C03569=1018.076,43.871,-109.128,166.538,54.047,159.849
C03570=1018.081,44.120,-109.143,166.541,54.040,159.848
C03571=1018.087,44.370,-109.159,166.544,54.032,159.847
C03572=1018.092,44.619,-109.174,166.546,54.025,159.846
C03573=1018.097,44.868,-109.190,166.549,54.018,159.846
C03574=1018.102,45.118,-109.206,166.552,54.011,159.845
C03575=1018.107,45.367,-109.221,166.553,54.004,159.844
C03576=1018.113,45.617,-109.237,166.556,53.997,159.843
C03577=1018.118,45.867,-109.252,166.559,53.989,159.842
C03578=1018.123,46.116,-109.267,166.561,53.982,159.841
C03579=1018.129,46.365,-109.283,166.564,53.975,159.841
C03580=1018.134,46.615,-109.298,166.567,53.968,159.840
C03581=1018.140,46.865,-109.314,166.569,53.961,159.839
C03582=1018.145,47.114,-109.329,166.572,53.954,159.838
C03583=1018.150,47.364,-109.345,166.575,53.946,159.837
C03584=1018.156,47.612,-109.361,166.577,53.939,159.836
C03585=1018.161,47.862,-109.376,166.580,53.932,159.836
C03586=1018.166,48.112,-109.391,166.582,53.925,159.835
C03587=1018.171,48.361,-109.406,166.584,53.918,159.834
C03588=1018.177,48.610,-109.423,166.587,53.911,159.833
C03589=1018.182,48.860,-109.438,166.590,53.903,159.832
C03590=1018.188,49.110,-109.453,166.592,53.896,159.831
C03591=1018.193,49.359,-109.469,166.595,53.889,159.831
C03592=1018.199,49.608,-109.485,166.598,53.882,159.830
C03593=1018.203,49.858,-109.501,166.600,53.875,159.829
C03594=1018.209,50.108,-109.516,166.603,53.868,159.828
C03595=1018.214,50.357,-109.531,166.606,53.860,159.827
C03596=1018.220,50.606,-109.548,166.609,53.853,159.827
C03597=1018.225,50.856,-109.563,166.611,53.846,159.826
C03598=1018.231,51.106,-109.578,166.613,53.839,159.825
C03599=1018.236,51.354,-109.594,166.616,53.832,159.824
C03600=1018.242,51.604,-109.610,166.618,53.825,159.823
C03601=1018.247,51.853,-109.625,166.621,53.817,159.822
C03602=1018.253,52.103,-109.641,166.624,53.810,159.821
C03603=1018.258,52.352,-109.656,166.626,53.803,159.820
C03604=1018.263,52.602,-109.672,166.629,53.795,159.820
C03605=1018.268,52.851,-109.687,166.632,53.788,159.819
C03606=1018.274,53.101,-109.703,166.634,53.781,159.818
C03607=1018.279,53.350,-109.719,166.636,53.774,159.817
C03608=1018.285,53.600,-109.735,166.639,53.767,159.816
C03609=1018.290,53.849,-109.751,166.642,53.759,159.815
C03610=1018.295,54.099,-109.766,166.645,53.752,159.815
C03611=1018.301,54.347,-109.782,166.647,53.745,159.814
C03612=1018.306,54.597,-109.798,166.650,53.737,159.813
C03613=1018.312,54.847,-109.813,166.653,53.730,159.812
C03614=1018.317,55.096,-109.829,166.655,53.723,159.811
C03615=1018.323,55.346,-109.845,166.657,53.715,159.810
C03616=1018.328,55.595,-109.860,166.660,53.708,159.809
C03617=1018.334,55.845,-109.876,166.663,53.701,159.809
C03618=1018.339,56.094,-109.891,166.665,53.694,159.808
C03619=1018.345,56.343,-109.907,166.668,53.687,159.807
C03620=1018.351,56.593,-109.923,166.670,53.679,159.806
C03621=1018.356,56.842,-109.939,166.673,53.671,159.805
C03622=1018.361,57.092,-109.955,166.675,53.665,159.804
C03623=1018.366,57.341,-109.971,166.678,53.657,159.803
C03624=1018.372,57.591,-109.986,166.681,53.650,159.803
C03625=1018.377,57.841,-110.002,166.684,53.642,159.802
C03626=1018.383,58.089,-110.018,166.687,53.635,159.801
C03627=1018.388,58.339,-110.033,166.689,53.628,159.800
C03628=1018.395,58.621,-110.051,166.692,53.620,159.799
C03629=1018.401,58.904,-110.069,166.694,53.611,159.798
C03630=1018.407,59.186,-110.088,166.698,53.603,159.797
C03631=1018.413,59.469,-110.105,166.700,53.595,159.796
C03632=1018.419,59.718,-110.121,166.703,53.587,159.795
C03633=1018.425,59.968,-110.137,166.706,53.580,159.794
C03634=1018.430,60.217,-110.153,166.709,53.572,159.793
C03635=1018.436,60.467,-110.168,166.712,53.565,159.792
C03636=1018.441,60.715,-110.184,166.714,53.558,159.792
C03637=1018.447,60.965,-110.200,166.716,53.550,159.791
C03638=1018.453,61.215,-110.216,166.719,53.543,159.790
C03639=1018.458,61.464,-110.231,166.722,53.536,159.789
C03640=1018.463,61.714,-110.248,166.725,53.528,159.788
C03641=1018.469,61.964,-110.263,166.727,53.521,159.787
C03642=1018.474,62.213,-110.280,166.730,53.514,159.786
C03643=1018.480,62.462,-110.296,166.732,53.506,159.785
C03644=1018.485,62.712,-110.311,166.735,53.499,159.784
C03645=1018.491,62.961,-110.327,166.738,53.491,159.784
C03646=1018.496,63.211,-110.343,166.740,53.485,159.783
C03647=1018.502,63.460,-110.359,166.743,53.477,159.782
C03648=1018.507,63.701,-110.376,166.745,53.470,159.781
C03649=1018.512,63.942,-110.391,166.748,53.463,159.780
C03650=1018.518,64.183,-110.407,166.750,53.456,159.779
C03651=1018.523,64.424,-110.422,166.753,53.449,159.779
C03652=1018.528,64.666,-110.438,166.756,53.442,159.778
C03653=1018.533,64.907,-110.454,166.758,53.435,159.777
C03654=1018.539,65.148,-110.469,166.761,53.428,159.776
C03655=1018.543,65.389,-110.485,166.763,53.421,159.775
C03656=1018.549,65.638,-110.501,166.766,53.414,159.774
C03657=1018.554,65.888,-110.518,166.768,53.407,159.773
C03658=1018.560,66.137,-110.534,166.770,53.399,159.772
C03659=1018.565,66.387,-110.550,166.773,53.392,159.772
C03660=1018.571,66.636,-110.566,166.777,53.385,159.771
C03661=1018.576,66.885,-110.582,166.778,53.378,159.770
C03662=1018.581,67.135,-110.599,166.781,53.371,159.769
C03663=1018.587,67.384,-110.615,166.785,53.363,159.768
C03664=1018.592,67.634,-110.631,166.786,53.356,159.767
C03665=1018.597,67.883,-110.647,166.789,53.349,159.766
C03666=1018.603,68.133,-110.664,166.792,53.342,159.766
C03667=1018.609,68.382,-110.680,166.795,53.334,159.765
C03668=1018.614,68.632,-110.697,166.797,53.327,159.764
C03669=1018.619,68.880,-110.713,166.800,53.320,159.763
C03670=1018.624,69.130,-110.730,166.803,53.312,159.762
C03671=1018.630,69.380,-110.747,166.805,53.306,159.761
C03672=1018.635,69.629,-110.763,166.808,53.298,159.761
C03673=1018.640,69.878,-110.779,166.811,53.291,159.760
C03674=1018.646,70.127,-110.796,166.813,53.284,159.759
C03675=1018.651,70.377,-110.813,166.816,53.277,159.758
C03676=1018.656,70.627,-110.829,166.818,53.269,159.757
C03677=1018.662,70.876,-110.846,166.820,53.262,159.756
C03678=1018.667,71.125,-110.862,166.823,53.255,159.755
C03679=1018.673,71.374,-110.878,166.826,53.248,159.755
C03680=1018.678,71.624,-110.895,166.828,53.241,159.754
C03681=1018.683,71.874,-110.912,166.831,53.234,159.753
C03682=1018.689,72.123,-110.928,166.834,53.226,159.752
C03683=1018.694,72.372,-110.945,166.836,53.219,159.751
C03684=1018.699,72.621,-110.962,166.839,53.212,159.750
C03685=1018.705,72.871,-110.978,166.842,53.205,159.749
C03686=1018.710,73.120,-110.995,166.845,53.198,159.749
C03687=1018.716,73.370,-111.012,166.847,53.190,159.747
C03688=1018.721,73.619,-111.028,166.850,53.183,159.747
C03689=1018.726,73.868,-111.044,166.853,53.176,159.746
C03690=1018.732,74.118,-111.061,166.855,53.169,159.745
C03691=1018.737,74.367,-111.078,166.858,53.162,159.744
C03692=1018.743,74.666,-111.098,166.861,53.153,159.743
C03693=1018.750,74.965,-111.118,166.864,53.144,159.742
C03694=1018.756,75.265,-111.138,166.868,53.136,159.741
C03695=1018.763,75.563,-111.158,166.871,53.127,159.740
C03696=1018.768,75.813,-111.175,166.873,53.120,159.739
C03697=1018.774,76.062,-111.191,166.876,53.112,159.738
C03698=1018.780,76.312,-111.208,166.879,53.105,159.737
C03699=1018.785,76.560,-111.225,166.881,53.098,159.736
C03700=1018.790,76.810,-111.242,166.884,53.091,159.736
C03701=1018.796,77.059,-111.258,166.887,53.084,159.735
C03702=1018.801,77.309,-111.275,166.888,53.076,159.734
C03703=1018.806,77.559,-111.292,166.891,53.069,159.733
C03704=1018.812,77.808,-111.309,166.894,53.062,159.732
C03705=1018.817,78.057,-111.326,166.897,53.055,159.731
C03706=1018.822,78.307,-111.343,166.900,53.048,159.730
C03707=1018.828,78.556,-111.360,166.903,53.041,159.730
C03708=1018.832,78.805,-111.377,166.905,53.034,159.729
C03709=1018.837,79.055,-111.394,166.908,53.027,159.728
C03710=1018.843,79.304,-111.411,166.910,53.019,159.727
C03711=1018.848,79.553,-111.428,166.912,53.012,159.726
C03712=1018.854,79.803,-111.444,166.915,53.005,159.725
C03713=1018.860,80.052,-111.462,166.919,52.998,159.725
C03714=1018.865,80.301,-111.479,166.921,52.991,159.724
C03715=1018.870,80.551,-111.496,166.924,52.984,159.723
C03716=1018.876,80.800,-111.513,166.927,52.977,159.722
C03717=1018.881,81.050,-111.530,166.928,52.969,159.721
C03718=1018.886,81.299,-111.547,166.931,52.962,159.720
C03719=1018.891,81.548,-111.564,166.934,52.955,159.719
C03720=1018.896,81.797,-111.581,166.937,52.948,159.718
C03721=1018.902,82.046,-111.599,166.940,52.941,159.718
C03722=1018.907,82.296,-111.615,166.942,52.933,159.717
C03723=1018.912,82.546,-111.632,166.944,52.927,159.716
C03724=1018.918,82.795,-111.650,166.947,52.919,159.715
C03725=1018.923,83.044,-111.667,166.950,52.912,159.714
C03726=1018.928,83.293,-111.684,166.953,52.905,159.713
C03727=1018.934,83.543,-111.701,166.955,52.898,159.712
C03728=1018.939,83.792,-111.717,166.958,52.890,159.712
C03729=1018.945,84.041,-111.735,166.961,52.883,159.711
C03730=1018.950,84.291,-111.752,166.963,52.877,159.710
C03731=1018.956,84.540,-111.769,166.966,52.869,159.709
C03732=1018.961,84.790,-111.786,166.969,52.862,159.708
C03733=1018.966,85.039,-111.804,166.971,52.855,159.707
C03734=1018.972,85.289,-111.821,166.974,52.848,159.706
C03735=1018.977,85.538,-111.838,166.977,52.840,159.705
C03736=1018.982,85.787,-111.855,166.980,52.833,159.705
C03737=1018.988,86.036,-111.873,166.982,52.826,159.704
C03738=1018.993,86.286,-111.890,166.985,52.819,159.703
C03739=1018.998,86.536,-111.906,166.988,52.811,159.702
C03740=1019.004,86.785,-111.924,166.990,52.804,159.701
C03741=1019.009,87.034,-111.941,166.993,52.797,159.700
C03742=1019.015,87.283,-111.958,166.996,52.789,159.699
C03743=1019.020,87.532,-111.976,166.999,52.782,159.698
C03744=1019.025,87.782,-111.993,167.001,52.775,159.698
C03745=1019.032,88.031,-112.010,167.004,52.768,159.697
C03746=1019.037,88.280,-112.027,167.007,52.760,159.696
C03747=1019.042,88.529,-112.044,167.010,52.753,159.695
C03748=1019.048,88.779,-112.061,167.012,52.747,159.694
C03749=1019.053,89.028,-112.079,167.015,52.739,159.693
C03750=1019.058,89.278,-112.096,167.018,52.732,159.692
C03751=1019.064,89.528,-112.114,167.021,52.725,159.692
C03752=1019.069,89.777,-112.132,167.023,52.718,159.691
C03753=1019.074,90.027,-112.148,167.026,52.711,159.690
C03754=1019.079,90.276,-112.167,167.029,52.703,159.689
C03755=1019.085,90.525,-112.184,167.031,52.696,159.688
C03756=1019.091,90.807,-112.204,167.034,52.688,159.687
C03757=1019.097,91.090,-112.224,167.037,52.680,159.686
C03758=1019.102,91.373,-112.244,167.040,52.672,159.685
C03759=1019.108,91.654,-112.263,167.044,52.664,159.684
C03760=1019.115,91.904,-112.281,167.047,52.657,159.683
C03761=1019.119,92.154,-112.299,167.048,52.650,159.682
C03762=1019.125,92.403,-112.317,167.051,52.642,159.682
C03763=1019.130,92.652,-112.333,167.055,52.635,159.681
C03764=1019.135,92.902,-112.352,167.057,52.629,159.680
C03765=1019.140,93.151,-112.369,167.060,52.622,159.679
C03766=1019.146,93.400,-112.387,167.063,52.614,159.678
C03767=1019.151,93.649,-112.404,167.065,52.607,159.677
C03768=1019.156,93.899,-112.422,167.068,52.600,159.676
C03769=1019.161,94.148,-112.439,167.071,52.593,159.676
C03770=1019.167,94.397,-112.457,167.074,52.585,159.675
C03771=1019.173,94.646,-112.475,167.076,52.578,159.674
C03772=1019.178,94.896,-112.493,167.079,52.571,159.673
C03773=1019.183,95.145,-112.510,167.082,52.564,159.672
C03774=1019.188,95.395,-112.527,167.084,52.557,159.671
C03775=1019.194,95.644,-112.545,167.087,52.550,159.670
C03776=1019.199,95.893,-112.563,167.090,52.542,159.669
C03777=1019.204,96.142,-112.581,167.093,52.535,159.669
C03778=1019.210,96.392,-112.599,167.095,52.528,159.668
C03779=1019.215,96.641,-112.617,167.098,52.521,159.667
C03780=1019.221,96.890,-112.634,167.101,52.514,159.666
C03781=1019.226,97.140,-112.651,167.104,52.507,159.665
C03782=1019.231,97.389,-112.669,167.106,52.499,159.664
C03783=1019.236,97.638,-112.687,167.109,52.492,159.663
C03784=1019.242,97.888,-112.705,167.112,52.485,159.663
C03785=1019.248,98.137,-112.722,167.115,52.477,159.662
C03786=1019.253,98.386,-112.740,167.117,52.471,159.661
C03787=1019.258,98.635,-112.758,167.120,52.464,159.660
C03788=1019.264,98.884,-112.776,167.123,52.456,159.659
C03789=1019.270,99.134,-112.794,167.126,52.449,159.658
C03790=1019.275,99.383,-112.812,167.128,52.442,159.657
C03791=1019.280,99.632,-112.829,167.131,52.435,159.656
C03792=1019.285,99.882,-112.848,167.135,52.428,159.656
C03793=1019.290,100.131,-112.865,167.137,52.421,159.655
C03794=1019.296,100.381,-112.884,167.139,52.413,159.654
C03795=1019.301,100.630,-112.902,167.143,52.406,159.653
C03796=1019.306,100.879,-112.919,167.145,52.400,159.652
C03797=1019.311,101.129,-112.938,167.148,52.393,159.651
C03798=1019.316,101.378,-112.955,167.151,52.385,159.651
C03799=1019.322,101.627,-112.974,167.153,52.378,159.649
C03800=1019.328,101.876,-112.992,167.156,52.371,159.649
C03801=1019.332,102.126,-113.010,167.159,52.364,159.648
C03802=1019.337,102.375,-113.028,167.162,52.357,159.647
C03803=1019.343,102.625,-113.046,167.164,52.350,159.646
C03804=1019.348,102.874,-113.064,167.168,52.343,159.645
C03805=1019.354,103.123,-113.082,167.170,52.335,159.644
C03806=1019.359,103.372,-113.101,167.172,52.329,159.643
C03807=1019.365,103.621,-113.119,167.176,52.322,159.643
C03808=1019.370,103.871,-113.137,167.179,52.315,159.642
C03809=1019.374,104.120,-113.155,167.182,52.307,159.641
C03810=1019.380,104.369,-113.173,167.184,52.300,159.640
C03811=1019.385,104.619,-113.191,167.187,52.293,159.639
C03812=1019.391,104.868,-113.209,167.190,52.286,159.638
C03813=1019.396,105.117,-113.228,167.192,52.279,159.637
C03814=1019.401,105.366,-113.245,167.195,52.272,159.637
C03815=1019.407,105.616,-113.264,167.198,52.264,159.636
C03816=1019.412,105.865,-113.283,167.201,52.257,159.635
C03817=1019.417,106.114,-113.300,167.203,52.250,159.634
C03818=1019.423,106.364,-113.319,167.206,52.243,159.633
C03819=1019.428,106.613,-113.336,167.209,52.236,159.632
C03820=1019.434,106.895,-113.357,167.212,52.228,159.631
C03821=1019.441,107.178,-113.378,167.216,52.219,159.630
C03822=1019.447,107.461,-113.398,167.219,52.211,159.629
C03823=1019.453,107.743,-113.419,167.222,52.204,159.628
C03824=1019.458,107.993,-113.438,167.225,52.197,159.628
C03825=1019.463,108.242,-113.456,167.228,52.189,159.627
C03826=1019.468,108.491,-113.473,167.230,52.182,159.626
C03827=1019.474,108.741,-113.493,167.234,52.175,159.625
C03828=1019.480,108.990,-113.510,167.236,52.167,159.624
C03829=1019.484,109.239,-113.528,167.239,52.160,159.623
C03830=1019.491,109.488,-113.547,167.243,52.153,159.622
C03831=1019.495,109.737,-113.565,167.245,52.147,159.622
C03832=1019.500,109.987,-113.583,167.248,52.139,159.621
C03833=1019.506,110.236,-113.603,167.251,52.132,159.620
C03834=1019.511,110.486,-113.621,167.254,52.125,159.619
C03835=1019.517,110.734,-113.639,167.256,52.118,159.618
C03836=1019.522,110.984,-113.658,167.259,52.110,159.617
C03837=1019.527,111.233,-113.676,167.262,52.103,159.616
C03838=1019.532,111.482,-113.695,167.265,52.096,159.616
C03839=1019.538,111.732,-113.713,167.268,52.090,159.615
C03840=1019.543,111.981,-113.731,167.270,52.082,159.614
C03841=1019.548,112.231,-113.750,167.274,52.075,159.613
C03842=1019.553,112.479,-113.769,167.277,52.068,159.612
C03843=1019.558,112.729,-113.787,167.279,52.061,159.611
C03844=1019.564,112.978,-113.806,167.282,52.054,159.610
C03845=1019.569,113.227,-113.825,167.285,52.047,159.610
C03846=1019.574,113.477,-113.844,167.288,52.041,159.609
C03847=1019.580,113.726,-113.863,167.291,52.034,159.608
C03848=1019.585,113.974,-113.881,167.294,52.027,159.607
C03849=1019.590,114.224,-113.900,167.296,52.019,159.606
C03850=1019.595,114.473,-113.919,167.299,52.012,159.605
C03851=1019.600,114.722,-113.938,167.302,52.005,159.605
C03852=1019.606,114.972,-113.956,167.305,51.999,159.604
C03853=1019.611,115.221,-113.975,167.308,51.992,159.603
C03854=1019.616,115.470,-113.995,167.311,51.985,159.602
C03855=1019.620,115.720,-114.013,167.314,51.978,159.601
C03856=1019.625,115.968,-114.032,167.316,51.971,159.600
C03857=1019.631,116.218,-114.051,167.319,51.963,159.599
C03858=1019.636,116.467,-114.069,167.322,51.956,159.599
C03859=1019.642,116.717,-114.089,167.325,51.950,159.598
C03860=1019.647,116.965,-114.107,167.328,51.943,159.597
C03861=1019.652,117.215,-114.126,167.331,51.936,159.596
C03862=1019.657,117.464,-114.145,167.334,51.929,159.595
C03863=1019.663,117.714,-114.164,167.336,51.921,159.594
C03864=1019.668,117.962,-114.183,167.339,51.914,159.594
C03865=1019.673,118.212,-114.201,167.343,51.907,159.593
C03866=1019.678,118.461,-114.220,167.346,51.900,159.592
C03867=1019.683,118.710,-114.239,167.348,51.894,159.591
C03868=1019.689,118.959,-114.259,167.351,51.887,159.590
C03869=1019.694,119.209,-114.277,167.354,51.879,159.589
C03870=1019.699,119.458,-114.297,167.357,51.872,159.589
C03871=1019.704,119.707,-114.315,167.360,51.865,159.588
C03872=1019.710,119.957,-114.335,167.363,51.858,159.587
C03873=1019.715,120.205,-114.354,167.366,51.851,159.586
C03874=1019.720,120.455,-114.372,167.369,51.844,159.585
C03875=1019.725,120.704,-114.391,167.372,51.837,159.584
C03876=1019.731,120.954,-114.410,167.374,51.830,159.583
C03877=1019.736,121.202,-114.429,167.378,51.823,159.583
C03878=1019.742,121.452,-114.448,167.381,51.815,159.582
C03879=1019.747,121.700,-114.467,167.384,51.808,159.581
C03880=1019.752,121.950,-114.486,167.387,51.801,159.580
C03881=1019.757,122.199,-114.505,167.389,51.795,159.579
C03882=1019.763,122.449,-114.524,167.393,51.788,159.578
C03883=1019.768,122.697,-114.543,167.395,51.780,159.577
C03884=1019.774,122.980,-114.565,167.399,51.772,159.577
C03885=1019.780,123.263,-114.587,167.402,51.764,159.576
C03886=1019.786,123.545,-114.608,167.406,51.756,159.575
C03887=1019.792,123.828,-114.630,167.408,51.748,159.574
C03888=1019.798,124.078,-114.649,167.412,51.741,159.573
C03889=1019.803,124.326,-114.668,167.415,51.734,159.572
C03890=1019.808,124.576,-114.687,167.418,51.727,159.571
C03891=1019.814,124.824,-114.706,167.421,51.719,159.570
C03892=1019.819,125.074,-114.724,167.424,51.713,159.569
C03893=1019.824,125.323,-114.743,167.427,51.706,159.569
C03894=1019.830,125.573,-114.762,167.430,51.698,159.568
C03895=1019.835,125.822,-114.782,167.433,51.691,159.567
C03896=1019.840,126.071,-114.801,167.436,51.684,159.566
C03897=1019.845,126.321,-114.820,167.439,51.677,159.565
C03898=1019.850,126.569,-114.839,167.442,51.670,159.564
C03899=1019.856,126.819,-114.859,167.445,51.663,159.563
C03900=1019.862,127.068,-114.878,167.449,51.656,159.563
C03901=1019.867,127.317,-114.897,167.451,51.648,159.562
C03902=1019.873,127.566,-114.916,167.454,51.642,159.561
C03903=1019.878,127.816,-114.935,167.457,51.635,159.560
C03904=1019.883,128.064,-114.954,167.460,51.627,159.559
C03905=1019.889,128.314,-114.973,167.463,51.620,159.558
C03906=1019.894,128.564,-114.993,167.467,51.613,159.557
C03907=1019.899,128.812,-115.012,167.469,51.605,159.557
C03908=1019.905,129.062,-115.031,167.473,51.598,159.556
C03909=1019.910,129.311,-115.050,167.476,51.592,159.555
C03910=1019.916,129.560,-115.069,167.479,51.584,159.554
C03911=1019.921,129.809,-115.089,167.482,51.577,159.553
C03912=1019.927,130.059,-115.108,167.485,51.570,159.552
C03913=1019.932,130.307,-115.128,167.488,51.563,159.552
C03914=1019.937,130.557,-115.147,167.491,51.556,159.551
C03915=1019.942,130.806,-115.167,167.494,51.549,159.550
C03916=1019.947,131.055,-115.186,167.497,51.542,159.549
C03917=1019.952,131.305,-115.206,167.500,51.535,159.548
C03918=1019.958,131.554,-115.226,167.503,51.528,159.547
C03919=1019.963,131.803,-115.245,167.506,51.521,159.547
C03920=1019.968,132.052,-115.264,167.509,51.514,159.546
C03921=1019.974,132.301,-115.284,167.512,51.507,159.545
C03922=1019.979,132.550,-115.304,167.516,51.500,159.544
C03923=1019.984,132.799,-115.323,167.519,51.493,159.543
C03924=1019.989,133.049,-115.343,167.521,51.486,159.542
C03925=1019.995,133.297,-115.363,167.524,51.479,159.541
C03926=1020.000,133.547,-115.382,167.527,51.472,159.541
C03927=1020.005,133.797,-115.402,167.531,51.465,159.540
C03928=1020.011,134.045,-115.422,167.534,51.458,159.539
C03929=1020.016,134.294,-115.441,167.537,51.451,159.538
C03930=1020.021,134.544,-115.460,167.540,51.443,159.537
C03931=1020.027,134.793,-115.481,167.543,51.437,159.536
C03932=1020.032,135.042,-115.500,167.546,51.430,159.536
C03933=1020.037,135.291,-115.520,167.549,51.423,159.535
C03934=1020.043,135.540,-115.540,167.553,51.416,159.534
C03935=1020.048,135.790,-115.559,167.555,51.409,159.533
C03936=1020.053,136.039,-115.578,167.559,51.402,159.532
C03937=1020.058,136.288,-115.599,167.562,51.395,159.531
C03938=1020.064,136.537,-115.618,167.565,51.388,159.531
C03939=1020.069,136.786,-115.639,167.569,51.381,159.530
C03940=1020.074,137.035,-115.658,167.571,51.374,159.529
C03941=1020.079,137.284,-115.678,167.574,51.367,159.528
C03942=1020.085,137.534,-115.697,167.577,51.360,159.527
C03943=1020.090,137.783,-115.718,167.581,51.353,159.527
C03944=1020.096,138.032,-115.737,167.584,51.346,159.526
C03945=1020.100,138.281,-115.757,167.587,51.338,159.525
C03946=1020.105,138.530,-115.777,167.590,51.331,159.524
C03947=1020.111,138.780,-115.798,167.593,51.325,159.523
C03948=1020.117,139.062,-115.820,167.596,51.317,159.522
C03949=1020.123,139.345,-115.842,167.600,51.309,159.521
C03950=1020.129,139.627,-115.865,167.604,51.301,159.520
C03951=1020.135,139.910,-115.888,167.607,51.293,159.519
C03952=1020.140,140.158,-115.907,167.611,51.287,159.519
C03953=1020.145,140.408,-115.928,167.614,51.280,159.518
C03954=1020.150,140.657,-115.948,167.617,51.273,159.517
C03955=1020.155,140.906,-115.968,167.620,51.265,159.516
C03956=1020.161,141.155,-115.988,167.624,51.258,159.515
C03957=1020.166,141.404,-116.008,167.627,51.251,159.515
C03958=1020.171,141.653,-116.028,167.630,51.245,159.514
C03959=1020.177,141.902,-116.048,167.634,51.238,159.513
C03960=1020.182,142.152,-116.068,167.636,51.231,159.512
C03961=1020.187,142.401,-116.088,167.639,51.224,159.511
C03962=1020.192,142.650,-116.109,167.642,51.217,159.510
C03963=1020.197,142.899,-116.128,167.646,51.210,159.510
C03964=1020.203,143.148,-116.148,167.649,51.203,159.509
C03965=1020.208,143.397,-116.169,167.652,51.196,159.508
C03966=1020.214,143.646,-116.189,167.656,51.189,159.507
C03967=1020.219,143.896,-116.209,167.659,51.182,159.506
C03968=1020.224,144.145,-116.229,167.662,51.175,159.506
C03969=1020.229,144.394,-116.250,167.665,51.168,159.505
C03970=1020.235,144.643,-116.269,167.669,51.161,159.504
C03971=1020.240,144.893,-116.290,167.672,51.154,159.503
C03972=1020.245,145.141,-116.310,167.675,51.147,159.502
C03973=1020.251,145.390,-116.330,167.678,51.140,159.501
C03974=1020.256,145.640,-116.350,167.682,51.133,159.501
C03975=1020.261,145.889,-116.370,167.685,51.126,159.500
C03976=1020.266,146.138,-116.391,167.688,51.119,159.499
C03977=1020.272,146.387,-116.411,167.692,51.112,159.498
C03978=1020.277,146.636,-116.432,167.695,51.105,159.498
C03979=1020.282,146.885,-116.452,167.697,51.099,159.497
C03980=1020.288,147.134,-116.472,167.700,51.091,159.496
C03981=1020.293,147.384,-116.492,167.704,51.084,159.495
C03982=1020.298,147.633,-116.513,167.707,51.077,159.494
C03983=1020.304,147.882,-116.533,167.710,51.071,159.493
C03984=1020.309,148.131,-116.554,167.714,51.064,159.493
C03985=1020.314,148.379,-116.574,167.717,51.057,159.492
C03986=1020.319,148.629,-116.595,167.721,51.050,159.491
C03987=1020.324,148.878,-116.615,167.724,51.043,159.490
C03988=1020.329,149.127,-116.636,167.727,51.036,159.489
C03989=1020.335,149.376,-116.656,167.731,51.029,159.489
C03990=1020.340,149.625,-116.677,167.734,51.022,159.488
C03991=1020.345,149.874,-116.697,167.737,51.016,159.487
C03992=1020.350,150.123,-116.718,167.740,51.008,159.486
C03993=1020.356,150.372,-116.739,167.744,51.001,159.485
C03994=1020.361,150.622,-116.759,167.747,50.994,159.485
C03995=1020.366,150.871,-116.780,167.751,50.988,159.484
C03996=1020.371,151.120,-116.800,167.754,50.981,159.483
C03997=1020.377,151.369,-116.821,167.757,50.974,159.482
C03998=1020.382,151.618,-116.841,167.761,50.967,159.481
C03999=1020.387,151.867,-116.862,167.764,50.960,159.481
C04000=1020.392,152.116,-116.882,167.767,50.953,159.480
C04001=1020.398,152.365,-116.903,167.771,50.946,159.479
C04002=1020.403,152.614,-116.924,167.774,50.939,159.478
C04003=1020.408,152.863,-116.945,167.777,50.932,159.477
C04004=1020.414,153.112,-116.965,167.781,50.925,159.477
C04005=1020.419,153.361,-116.986,167.784,50.918,159.476
C04006=1020.424,153.610,-117.006,167.787,50.912,159.475
C04007=1020.429,153.860,-117.028,167.791,50.905,159.474
C04008=1020.434,154.109,-117.048,167.794,50.898,159.473
C04009=1020.440,154.358,-117.070,167.798,50.891,159.473
C04010=1020.445,154.607,-117.090,167.801,50.884,159.472
C04011=1020.451,154.857,-117.111,167.804,50.877,159.471
C04012=1020.456,155.139,-117.135,167.807,50.870,159.470
C04013=1020.462,155.421,-117.158,167.811,50.862,159.469
C04014=1020.469,155.703,-117.182,167.815,50.854,159.468
C04015=1020.474,155.985,-117.205,167.819,50.846,159.467
C04016=1020.480,156.234,-117.226,167.823,50.839,159.467
C04017=1020.484,156.483,-117.247,167.826,50.833,159.466
C04018=1020.490,156.733,-117.268,167.830,50.826,159.465
C04019=1020.495,156.982,-117.289,167.833,50.819,159.464
C04020=1020.501,157.231,-117.310,167.837,50.812,159.464
C04021=1020.506,157.480,-117.330,167.840,50.805,159.463
C04022=1020.511,157.729,-117.351,167.843,50.799,159.462
C04023=1020.516,157.978,-117.373,167.847,50.792,159.461
C04024=1020.521,158.227,-117.393,167.850,50.785,159.460
C04025=1020.527,158.476,-117.414,167.853,50.777,159.459
C04026=1020.532,158.725,-117.435,167.857,50.771,159.459
C04027=1020.538,158.974,-117.456,167.860,50.764,159.458
C04028=1020.543,159.223,-117.478,167.864,50.758,159.457
C04029=1020.547,159.473,-117.499,167.867,50.751,159.457
C04030=1020.553,159.721,-117.520,167.871,50.744,159.456
C04031=1020.558,159.971,-117.542,167.874,50.737,159.455
C04032=1020.563,160.219,-117.563,167.877,50.730,159.454
C04033=1020.568,160.468,-117.585,167.881,50.724,159.453
C04034=1020.572,160.717,-117.606,167.885,50.717,159.453
C04035=1020.579,160.967,-117.628,167.888,50.711,159.452
C04036=1020.583,161.216,-117.649,167.892,50.704,159.451
C04037=1020.588,161.465,-117.671,167.895,50.697,159.451
C04038=1020.593,161.713,-117.692,167.898,50.690,159.450
C04039=1020.598,161.963,-117.713,167.902,50.683,159.449
C04040=1020.604,162.211,-117.734,167.906,50.677,159.448
C04041=1020.608,162.460,-117.756,167.909,50.671,159.448
C04042=1020.614,162.710,-117.778,167.912,50.664,159.447
C04043=1020.619,162.959,-117.799,167.916,50.657,159.446
C04044=1020.624,163.208,-117.821,167.919,50.650,159.445
C04045=1020.628,163.457,-117.842,167.923,50.643,159.444
C04046=1020.634,163.706,-117.863,167.927,50.637,159.444
C04047=1020.639,163.954,-117.885,167.930,50.630,159.443
C04048=1020.645,164.204,-117.906,167.933,50.624,159.442
C04049=1020.649,164.453,-117.928,167.937,50.617,159.442
C04050=1020.654,164.702,-117.950,167.940,50.610,159.441
C04051=1020.660,164.950,-117.971,167.944,50.603,159.440
C04052=1020.665,165.200,-117.992,167.947,50.597,159.439
C04053=1020.670,165.449,-118.014,167.951,50.590,159.439
C04054=1020.675,165.698,-118.036,167.954,50.584,159.438
C04055=1020.680,165.947,-118.057,167.958,50.577,159.437
C04056=1020.685,166.197,-118.079,167.961,50.570,159.436
C04057=1020.691,166.445,-118.100,167.965,50.563,159.435
C04058=1020.696,166.694,-118.122,167.969,50.556,159.435
C04059=1020.701,166.943,-118.143,167.973,50.549,159.434
C04060=1020.707,167.192,-118.166,167.977,50.543,159.433
C04061=1020.711,167.441,-118.187,167.980,50.537,159.433
C04062=1020.717,167.690,-118.208,167.983,50.530,159.432
C04063=1020.722,167.939,-118.230,167.987,50.523,159.431
C04064=1020.727,168.188,-118.252,167.990,50.516,159.430
C04065=1020.733,168.437,-118.273,167.994,50.509,159.430
C04066=1020.737,168.686,-118.295,167.997,50.503,159.429
C04067=1020.743,168.936,-118.317,168.001,50.496,159.428
C04068=1020.748,169.184,-118.338,168.005,50.490,159.427
C04069=1020.753,169.433,-118.360,168.009,50.483,159.427
C04070=1020.759,169.682,-118.382,168.012,50.476,159.426
C04071=1020.764,169.931,-118.403,168.016,50.469,159.425
C04072=1020.769,170.180,-118.425,168.019,50.462,159.424
C04073=1020.775,170.429,-118.447,168.023,50.456,159.424
C04074=1020.780,170.678,-118.469,168.026,50.449,159.423
C04075=1020.785,170.927,-118.491,168.030,50.442,159.422
C04076=1020.791,171.209,-118.515,168.034,50.435,159.421
C04077=1020.797,171.491,-118.540,168.038,50.427,159.420
C04078=1020.803,171.773,-118.564,168.042,50.420,159.420
C04079=1020.809,172.055,-118.589,168.047,50.412,159.419
C04080=1020.814,172.304,-118.611,168.050,50.405,159.418
C04081=1020.819,172.553,-118.632,168.055,50.399,159.417
C04082=1020.825,172.802,-118.655,168.058,50.392,159.417
C04083=1020.830,173.051,-118.676,168.062,50.385,159.416
C04084=1020.836,173.300,-118.698,168.065,50.378,159.415
C04085=1020.841,173.549,-118.720,168.069,50.372,159.414
C04086=1020.847,173.798,-118.742,168.073,50.365,159.414
C04087=1020.851,174.047,-118.764,168.077,50.358,159.413
C04088=1020.856,174.296,-118.785,168.080,50.351,159.412
C04089=1020.862,174.545,-118.807,168.084,50.344,159.411
C04090=1020.867,174.794,-118.829,168.087,50.338,159.411
C04091=1020.873,175.043,-118.851,168.092,50.331,159.410
C04092=1020.878,175.292,-118.872,168.095,50.324,159.409
C04093=1020.884,175.541,-118.895,168.099,50.318,159.408
C04094=1020.889,175.790,-118.917,168.102,50.311,159.408
C04095=1020.895,176.039,-118.939,168.107,50.304,159.407
C04096=1020.900,176.288,-118.961,168.110,50.297,159.406
C04097=1020.905,176.537,-118.983,168.114,50.290,159.405
C04098=1020.911,176.786,-119.004,168.117,50.284,159.405
C04099=1020.916,177.035,-119.026,168.122,50.277,159.404
C04100=1020.921,177.284,-119.048,168.126,50.271,159.403
C04101=1020.928,177.532,-119.071,168.129,50.264,159.402
C04102=1020.932,177.781,-119.093,168.133,50.257,159.402
C04103=1020.938,178.031,-119.115,168.137,50.250,159.401
C04104=1020.943,178.279,-119.136,168.141,50.243,159.400
C04105=1020.949,178.529,-119.158,168.144,50.237,159.399
C04106=1020.954,178.777,-119.181,168.149,50.230,159.399
C04107=1020.960,179.026,-119.202,168.153,50.223,159.398
C04108=1020.965,179.275,-119.224,168.156,50.217,159.397
C04109=1020.970,179.525,-119.247,168.161,50.210,159.397
C04110=1020.976,179.774,-119.268,168.164,50.203,159.396
C04111=1020.982,180.022,-119.291,168.168,50.196,159.395
C04112=1020.987,180.271,-119.313,168.172,50.189,159.394
C04113=1020.993,180.520,-119.334,168.176,50.183,159.394
C04114=1020.998,180.769,-119.357,168.179,50.176,159.393
C04115=1021.004,181.018,-119.379,168.183,50.169,159.392
C04116=1021.009,181.267,-119.401,168.187,50.163,159.392
C04117=1021.015,181.516,-119.423,168.191,50.156,159.391
C04118=1021.020,181.765,-119.446,168.195,50.149,159.390
C04119=1021.025,182.014,-119.468,168.199,50.142,159.389
C04120=1021.032,182.263,-119.490,168.202,50.136,159.389
C04121=1021.036,182.512,-119.513,168.206,50.130,159.388
C04122=1021.042,182.761,-119.536,168.211,50.123,159.387
C04123=1021.046,183.011,-119.558,168.215,50.116,159.387
C04124=1021.051,183.259,-119.581,168.218,50.110,159.386
C04125=1021.057,183.508,-119.604,168.222,50.103,159.385
C04126=1021.062,183.756,-119.626,168.226,50.097,159.384
C04127=1021.067,184.006,-119.649,168.230,50.090,159.384
C04128=1021.073,184.255,-119.672,168.234,50.084,159.383
C04129=1021.077,184.503,-119.694,168.238,50.077,159.382
C04130=1021.082,184.753,-119.718,168.241,50.071,159.382
C04131=1021.088,185.002,-119.741,168.245,50.065,159.381
C04132=1021.093,185.250,-119.762,168.250,50.058,159.381
C04133=1021.098,185.500,-119.786,168.253,50.052,159.380
C04134=1021.103,185.748,-119.809,168.257,50.045,159.379
C04135=1021.109,185.997,-119.832,168.261,50.039,159.378
C04136=1021.114,186.246,-119.854,168.265,50.032,159.378
C04137=1021.119,186.495,-119.877,168.269,50.026,159.377
C04138=1021.124,186.744,-119.900,168.273,50.019,159.376
C04139=1021.129,186.993,-119.923,168.278,50.013,159.376
C04140=1021.135,187.274,-119.949,168.282,50.005,159.375
C04141=1021.142,187.556,-119.974,168.286,49.998,159.374
C04142=1021.148,187.837,-120.000,168.291,49.991,159.374
C04143=1021.154,188.119,-120.026,168.295,49.983,159.373
C04144=1021.158,188.368,-120.049,168.299,49.977,159.372
C04145=1021.164,188.617,-120.072,168.304,49.970,159.371
C04146=1021.169,188.866,-120.095,168.307,49.964,159.371
C04147=1021.174,189.114,-120.118,168.311,49.958,159.370
C04148=1021.180,189.363,-120.141,168.316,49.951,159.369
C04149=1021.185,189.612,-120.164,168.319,49.945,159.369
C04150=1021.190,189.861,-120.188,168.323,49.938,159.368
C04151=1021.195,190.110,-120.210,168.328,49.932,159.367
C04152=1021.201,190.359,-120.233,168.331,49.925,159.367
C04153=1021.206,190.608,-120.256,168.335,49.919,159.366
C04154=1021.212,190.857,-120.279,168.340,49.912,159.365
C04155=1021.217,191.105,-120.302,168.344,49.906,159.365
C04156=1021.222,191.354,-120.325,168.347,49.900,159.364
C04157=1021.227,191.603,-120.348,168.352,49.893,159.363
C04158=1021.233,191.852,-120.371,168.356,49.887,159.363
C04159=1021.238,192.101,-120.395,168.360,49.881,159.362
C04160=1021.244,192.350,-120.418,168.364,49.874,159.361
C04161=1021.249,192.598,-120.440,168.368,49.867,159.361
C04162=1021.254,192.848,-120.464,168.373,49.861,159.360
C04163=1021.260,193.097,-120.487,168.376,49.854,159.359
C04164=1021.265,193.345,-120.510,168.380,49.848,159.359
C04165=1021.270,193.595,-120.533,168.385,49.841,159.358
C04166=1021.276,193.844,-120.556,168.389,49.835,159.357
C04167=1021.281,194.092,-120.579,168.393,49.828,159.357
C04168=1021.286,194.341,-120.602,168.397,49.822,159.356
C04169=1021.292,194.589,-120.626,168.401,49.815,159.355
C04170=1021.298,194.838,-120.649,168.406,49.809,159.355
C04171=1021.303,195.087,-120.672,168.409,49.802,159.354
C04172=1021.309,195.336,-120.695,168.414,49.796,159.353
C04173=1021.314,195.585,-120.718,168.418,49.790,159.353
C04174=1021.319,195.834,-120.742,168.423,49.783,159.352
C04175=1021.325,196.083,-120.765,168.426,49.777,159.351
C04176=1021.330,196.332,-120.788,168.431,49.770,159.351
C04177=1021.336,196.580,-120.812,168.435,49.764,159.350
C04178=1021.341,196.829,-120.835,168.439,49.758,159.350
C04179=1021.346,197.078,-120.858,168.443,49.751,159.349
C04180=1021.352,197.327,-120.881,168.447,49.745,159.348
C04181=1021.358,197.576,-120.904,168.452,49.738,159.348
C04182=1021.363,197.825,-120.928,168.456,49.732,159.347
C04183=1021.369,198.073,-120.951,168.460,49.725,159.346
C04184=1021.375,198.322,-120.974,168.464,49.719,159.346
C04185=1021.380,198.572,-120.998,168.469,49.712,159.345
C04186=1021.386,198.820,-121.021,168.473,49.706,159.344
C04187=1021.391,199.069,-121.044,168.477,49.699,159.344
C04188=1021.396,199.318,-121.068,168.481,49.693,159.343
C04189=1021.402,199.566,-121.091,168.486,49.687,159.342
C04190=1021.407,199.815,-121.115,168.490,49.680,159.342
C04191=1021.412,200.065,-121.139,168.495,49.674,159.341
C04192=1021.418,200.313,-121.162,168.498,49.668,159.341
C04193=1021.423,200.562,-121.186,168.503,49.661,159.340
C04194=1021.429,200.811,-121.210,168.507,49.655,159.339
C04195=1021.434,201.060,-121.234,168.512,49.649,159.339
C04196=1021.440,201.308,-121.257,168.516,49.642,159.338
C04197=1021.445,201.557,-121.281,168.520,49.636,159.337
C04198=1021.450,201.806,-121.305,168.524,49.630,159.337
C04199=1021.456,202.054,-121.329,168.529,49.624,159.336
C04200=1021.461,202.303,-121.352,168.533,49.617,159.336
C04201=1021.467,202.553,-121.377,168.538,49.611,159.335
C04202=1021.472,202.802,-121.400,168.542,49.605,159.334
C04203=1021.478,203.050,-121.424,168.547,49.599,159.334
C04204=1021.506,204.302,-121.545,168.985,49.689,159.423
C04205=1021.511,204.516,-121.568,168.988,49.684,159.422
C04206=1021.516,204.731,-121.589,168.992,49.680,159.422
C04207=1021.522,204.946,-121.611,168.994,49.676,159.421
C04208=1021.528,205.161,-121.633,168.998,49.671,159.421
C04209=1021.533,205.376,-121.655,169.001,49.666,159.420
C04210=1021.538,205.591,-121.677,169.003,49.662,159.420
C04211=1021.543,205.805,-121.699,169.007,49.657,159.419
C04212=1021.550,206.055,-121.725,169.010,49.652,159.419
C04213=1021.556,206.303,-121.750,169.014,49.646,159.418
C04214=1021.563,206.552,-121.775,169.017,49.641,159.418
C04215=1021.569,206.800,-121.801,169.020,49.636,159.417
C04216=1021.575,207.049,-121.827,169.024,49.630,159.417
C04217=1021.582,207.297,-121.852,169.027,49.625,159.416
C04218=1021.588,207.546,-121.877,169.031,49.620,159.415
C04219=1021.594,207.795,-121.903,169.035,49.614,159.415
C04220=1021.601,208.043,-121.929,169.038,49.609,159.414
C04221=1021.606,208.292,-121.955,169.041,49.605,159.414
C04222=1021.612,208.540,-121.980,169.044,49.599,159.413
C04223=1021.619,208.789,-122.006,169.048,49.594,159.413
C04224=1021.626,209.038,-122.032,169.051,49.589,159.412
C04225=1021.632,209.287,-122.057,169.055,49.584,159.412
C04226=1021.638,209.535,-122.082,169.059,49.579,159.411
C04227=1021.644,209.783,-122.109,169.062,49.573,159.410
C04228=1021.650,210.032,-122.134,169.065,49.568,159.410
C04229=1021.656,210.280,-122.160,169.069,49.563,159.409
C04230=1021.663,210.529,-122.186,169.073,49.558,159.409
C04231=1021.669,210.778,-122.211,169.076,49.553,159.408
C04232=1021.675,211.027,-122.238,169.079,49.548,159.408
C04233=1021.681,211.275,-122.264,169.083,49.543,159.407
C04234=1021.688,211.523,-122.290,169.087,49.538,159.407
C04235=1021.693,211.772,-122.316,169.090,49.532,159.406
C04236=1021.700,212.020,-122.342,169.094,49.527,159.406
C04237=1021.706,212.269,-122.367,169.097,49.522,159.405
C04238=1021.712,212.517,-122.394,169.100,49.517,159.404
C04239=1021.719,212.767,-122.419,169.104,49.512,159.404
C04240=1021.725,213.015,-122.445,169.108,49.507,159.404
C04241=1021.731,213.264,-122.471,169.111,49.502,159.403
C04242=1021.737,213.512,-122.497,169.114,49.497,159.402
C04243=1021.743,213.761,-122.523,169.118,49.492,159.402
C04244=1021.750,214.010,-122.550,169.122,49.487,159.401
C04245=1021.756,214.258,-122.575,169.125,49.482,159.401
C04246=1021.763,214.506,-122.601,169.128,49.477,159.400
C04247=1021.768,214.755,-122.628,169.133,49.472,159.400
C04248=1021.775,215.004,-122.653,169.136,49.467,159.399
C04249=1021.782,215.252,-122.679,169.139,49.462,159.399
C04250=1021.787,215.501,-122.705,169.143,49.457,159.398
C04251=1021.794,215.749,-122.731,169.147,49.452,159.398
C04252=1021.800,215.997,-122.757,169.150,49.447,159.397
C04253=1021.806,216.247,-122.784,169.153,49.442,159.397
C04254=1021.813,216.495,-122.810,169.157,49.438,159.396
C04255=1021.819,216.743,-122.836,169.161,49.433,159.396
C04256=1021.825,216.993,-122.862,169.164,49.428,159.395
C04257=1021.832,217.241,-122.888,169.168,49.423,159.395
C04258=1021.838,217.489,-122.914,169.171,49.418,159.394
C04259=1021.844,217.738,-122.940,169.175,49.413,159.394
C04260=1021.851,217.987,-122.967,169.179,49.408,159.393
C04261=1021.857,218.235,-122.993,169.182,49.403,159.393
C04262=1021.863,218.484,-123.019,169.186,49.398,159.392
C04263=1021.869,218.732,-123.045,169.190,49.394,159.392
C04264=1021.875,218.949,-123.069,169.192,49.390,159.392
C04265=1021.880,219.166,-123.091,169.196,49.385,159.391
C04266=1021.886,219.383,-123.114,169.198,49.381,159.391
C04267=1021.891,219.600,-123.137,169.202,49.377,159.390
C04268=1021.896,219.817,-123.161,169.204,49.373,159.390
C04269=1021.901,220.034,-123.183,169.208,49.369,159.389
C04270=1021.907,220.251,-123.206,169.212,49.364,159.389
C04271=1021.913,220.468,-123.230,169.214,49.361,159.389
C04272=1021.919,220.717,-123.256,169.218,49.356,159.388
C04273=1021.925,220.965,-123.283,169.222,49.351,159.388
C04274=1021.932,221.214,-123.309,169.226,49.346,159.387
C04275=1021.937,221.462,-123.336,169.229,49.341,159.387
C04276=1021.944,221.710,-123.362,169.232,49.337,159.386
C04277=1021.950,221.959,-123.389,169.236,49.332,159.386
C04278=1021.956,222.207,-123.416,169.240,49.327,159.385
C04279=1021.963,222.456,-123.442,169.244,49.323,159.385
C04280=1021.969,222.705,-123.469,169.247,49.318,159.385
C04281=1021.975,222.953,-123.495,169.250,49.313,159.384
C04282=1021.982,223.202,-123.522,169.254,49.309,159.384
C04283=1021.988,223.450,-123.548,169.258,49.304,159.383
C04284=1021.993,223.698,-123.575,169.262,49.299,159.383
C04285=1022.001,223.947,-123.601,169.265,49.294,159.382
C04286=1022.006,224.196,-123.628,169.269,49.290,159.382
C04287=1022.013,224.445,-123.655,169.272,49.285,159.381
C04288=1022.019,224.693,-123.681,169.276,49.280,159.381
C04289=1022.026,224.942,-123.708,169.280,49.276,159.381
C04290=1022.032,225.190,-123.734,169.283,49.271,159.380
C04291=1022.038,225.438,-123.761,169.287,49.267,159.380
C04292=1022.044,225.687,-123.788,169.290,49.262,159.379
C04293=1022.051,225.935,-123.815,169.295,49.257,159.379
C04294=1022.057,226.184,-123.842,169.298,49.253,159.378
C04295=1022.063,226.432,-123.868,169.302,49.248,159.378
C04296=1022.070,226.681,-123.895,169.305,49.244,159.378
C04297=1022.076,226.929,-123.921,169.309,49.239,159.377
C04298=1022.083,227.178,-123.948,169.313,49.235,159.377
C04299=1022.089,227.426,-123.976,169.317,49.230,159.376
C04300=1022.094,227.674,-124.002,169.320,49.226,159.376
C04301=1022.101,227.923,-124.029,169.324,49.221,159.376
C04302=1022.108,228.171,-124.056,169.327,49.217,159.375
C04303=1022.114,228.420,-124.083,169.331,49.212,159.375
C04304=1022.120,228.668,-124.110,169.335,49.208,159.375
C04305=1022.126,228.917,-124.137,169.339,49.203,159.374
C04306=1022.132,229.165,-124.164,169.342,49.199,159.374
C04307=1022.139,229.414,-124.191,169.346,49.195,159.373
C04308=1022.144,229.662,-124.218,169.349,49.190,159.373
C04309=1022.151,229.911,-124.246,169.353,49.186,159.372
C04310=1022.157,230.159,-124.272,169.358,49.181,159.372
C04311=1022.164,230.407,-124.299,169.361,49.177,159.372
C04312=1022.171,230.656,-124.326,169.365,49.172,159.371
C04313=1022.176,230.905,-124.354,169.368,49.168,159.371
C04314=1022.182,231.154,-124.381,169.372,49.164,159.370
C04315=1022.188,231.402,-124.408,169.375,49.159,159.370
C04316=1022.195,231.650,-124.436,169.379,49.155,159.370
C04317=1022.200,231.899,-124.462,169.382,49.150,159.369
C04318=1022.207,232.147,-124.490,169.387,49.146,159.369
C04319=1022.213,232.396,-124.517,169.391,49.142,159.369
C04320=1022.220,232.644,-124.545,169.394,49.137,159.368
C04321=1022.225,232.892,-124.571,169.398,49.133,159.368
C04322=1022.232,233.141,-124.599,169.402,49.129,159.368
C04323=1022.239,233.389,-124.627,169.405,49.125,159.367
C04324=1022.244,233.602,-124.649,169.409,49.121,159.367
C04325=1022.249,233.815,-124.673,169.412,49.117,159.367
C04326=1022.254,234.028,-124.697,169.416,49.113,159.366
C04327=1022.260,234.241,-124.720,169.419,49.110,159.366
C04328=1022.265,234.455,-124.743,169.421,49.106,159.366
C04329=1022.271,234.667,-124.767,169.425,49.103,159.365
C04330=1022.277,234.880,-124.790,169.428,49.099,159.365
C04331=1022.281,235.093,-124.814,169.432,49.095,159.365
C04332=1022.288,235.342,-124.841,169.436,49.091,159.364
C04333=1022.294,235.590,-124.868,169.439,49.087,159.364
C04334=1022.300,235.838,-124.896,169.443,49.083,159.364
C04335=1022.307,236.087,-124.923,169.446,49.078,159.363
C04336=1022.313,236.335,-124.951,169.450,49.074,159.363
C04337=1022.320,236.584,-124.978,169.454,49.070,159.363
C04338=1022.326,236.833,-125.005,169.458,49.065,159.362
C04339=1022.332,237.080,-125.033,169.462,49.061,159.362
C04340=1022.339,237.329,-125.060,169.466,49.057,159.362
C04341=1022.345,237.578,-125.089,169.469,49.053,159.361
C04342=1022.350,237.826,-125.115,169.473,49.049,159.361
C04343=1022.357,238.074,-125.143,169.477,49.045,159.361
C04344=1022.364,238.323,-125.171,169.480,49.040,159.360
C04345=1022.370,238.571,-125.198,169.484,49.036,159.360
C04346=1022.376,238.820,-125.225,169.489,49.032,159.360
C04347=1022.383,239.068,-125.253,169.492,49.028,159.359
C04348=1022.390,239.317,-125.281,169.496,49.023,159.359
C04349=1022.395,239.565,-125.309,169.500,49.020,159.359
C04350=1022.402,239.813,-125.336,169.504,49.016,159.358
C04351=1022.408,240.061,-125.364,169.507,49.011,159.358
C04352=1022.414,240.309,-125.392,169.511,49.007,159.358
C04353=1022.420,240.558,-125.420,169.515,49.004,159.358
C04354=1022.426,240.807,-125.448,169.519,49.000,159.357
C04355=1022.433,241.055,-125.476,169.523,48.995,159.357
C04356=1022.439,241.303,-125.503,169.527,48.991,159.357
C04357=1022.445,241.552,-125.532,169.531,48.987,159.356
C04358=1022.452,241.800,-125.559,169.535,48.983,159.356
C04359=1022.458,242.049,-125.588,169.538,48.979,159.356
C04360=1022.464,242.297,-125.615,169.542,48.976,159.356
C04361=1022.470,242.545,-125.643,169.546,48.971,159.355
C04362=1022.476,242.794,-125.671,169.550,48.967,159.355
C04363=1022.483,243.042,-125.699,169.554,48.964,159.355
C04364=1022.489,243.291,-125.727,169.557,48.960,159.354
C04365=1022.495,243.539,-125.754,169.561,48.955,159.354
C04366=1022.501,243.787,-125.783,169.566,48.952,159.354
C04367=1022.508,244.035,-125.811,169.570,48.947,159.353
C04368=1022.514,244.284,-125.840,169.574,48.944,159.353
C04369=1022.519,244.532,-125.868,169.577,48.940,159.353
C04370=1022.526,244.780,-125.896,169.581,48.936,159.353
C04371=1022.532,245.029,-125.924,169.585,48.932,159.352
C04372=1022.538,245.277,-125.953,169.589,48.928,159.352
C04373=1022.545,245.525,-125.981,169.593,48.924,159.352
C04374=1022.550,245.773,-126.009,169.597,48.921,159.352
C04375=1022.556,246.022,-126.037,169.600,48.917,159.351
C04376=1022.563,246.270,-126.066,169.604,48.913,159.351
C04377=1022.569,246.519,-126.094,169.608,48.910,159.351
C04378=1022.575,246.767,-126.122,169.612,48.905,159.351
C04379=1022.582,247.015,-126.151,169.616,48.902,159.351
C04380=1022.588,247.263,-126.179,169.620,48.898,159.350
C04381=1022.594,247.512,-126.207,169.624,48.894,159.350
C04382=1022.601,247.760,-126.236,169.627,48.890,159.350
C04383=1022.607,248.009,-126.264,169.631,48.887,159.349
C04384=1022.617,248.429,-126.312,169.638,48.880,159.349
C04385=1022.627,248.848,-126.360,169.645,48.874,159.349
C04386=1022.638,249.268,-126.408,169.652,48.867,159.348
C04387=1022.649,249.688,-126.456,169.659,48.861,159.348
C04388=1022.655,249.936,-126.485,169.663,48.857,159.348
C04389=1022.662,250.184,-126.513,169.667,48.854,159.348
C04390=1022.668,250.432,-126.542,169.671,48.850,159.347
C04391=1022.674,250.681,-126.570,169.674,48.846,159.347
C04392=1022.680,250.929,-126.599,169.679,48.843,159.347
C04393=1022.687,251.178,-126.627,169.683,48.839,159.347
C04394=1022.693,251.426,-126.656,169.686,48.835,159.346
C04395=1022.699,251.674,-126.684,169.690,48.831,159.346
C04396=1022.706,251.922,-126.712,169.694,48.828,159.346
C04397=1022.712,252.170,-126.741,169.698,48.824,159.346
C04398=1022.718,252.419,-126.770,169.702,48.820,159.345
C04399=1022.725,252.667,-126.799,169.706,48.817,159.345
C04400=1022.731,252.916,-126.827,169.711,48.813,159.345
C04401=1022.738,253.164,-126.856,169.715,48.810,159.345
C04402=1022.744,253.412,-126.885,169.719,48.805,159.345
C04403=1022.751,253.660,-126.913,169.723,48.802,159.344
C04404=1022.757,253.909,-126.942,169.727,48.798,159.344
C04405=1022.763,254.157,-126.971,169.731,48.795,159.344
C04406=1022.770,254.405,-126.999,169.735,48.791,159.344
C04407=1022.776,254.653,-127.028,169.739,48.788,159.344
C04408=1022.782,254.901,-127.057,169.742,48.784,159.343
C04409=1022.789,255.149,-127.085,169.746,48.780,159.343
C04410=1022.795,255.398,-127.113,169.751,48.776,159.343
C04411=1022.801,255.646,-127.142,169.755,48.773,159.343
C04412=1022.808,255.894,-127.172,169.759,48.770,159.343
C04413=1022.815,256.143,-127.200,169.763,48.766,159.343
C04414=1022.821,256.392,-127.229,169.768,48.763,159.342
C04415=1022.827,256.640,-127.258,169.772,48.759,159.342
C04416=1022.834,256.887,-127.286,169.776,48.756,159.342
C04417=1022.841,257.136,-127.315,169.779,48.751,159.342
C04418=1022.847,257.384,-127.344,169.783,48.748,159.342
C04419=1022.853,257.632,-127.373,169.787,48.744,159.341
C04420=1022.861,257.881,-127.401,169.792,48.741,159.341
C04421=1022.867,258.129,-127.430,169.796,48.737,159.341
C04422=1022.873,258.377,-127.459,169.800,48.734,159.341
C04423=1022.880,258.625,-127.488,169.804,48.730,159.341
C04424=1022.886,258.873,-127.517,169.808,48.727,159.341
C04425=1022.892,259.121,-127.546,169.812,48.723,159.340
C04426=1022.899,259.370,-127.575,169.816,48.720,159.340
C04427=1022.906,259.618,-127.604,169.820,48.716,159.340
C04428=1022.913,259.866,-127.633,169.825,48.712,159.340
C04429=1022.919,260.114,-127.662,169.829,48.709,159.340
C04430=1022.926,260.362,-127.690,169.833,48.706,159.340
C04431=1022.933,260.611,-127.720,169.838,48.702,159.339
C04432=1022.938,260.859,-127.749,169.842,48.699,159.339
C04433=1022.944,261.107,-127.778,169.846,48.696,159.339
C04434=1022.951,261.356,-127.807,169.850,48.692,159.339
C04435=1022.957,261.604,-127.836,169.854,48.689,159.339
C04436=1022.964,261.852,-127.867,169.858,48.686,159.339
C04437=1022.970,262.100,-127.896,169.862,48.682,159.339
C04438=1022.977,262.348,-127.925,169.866,48.679,159.339
C04439=1022.983,262.596,-127.954,169.870,48.676,159.338
C04440=1022.993,263.014,-128.004,169.878,48.670,159.338
C04441=1023.005,263.433,-128.053,169.884,48.664,159.338
C04442=1023.015,263.851,-128.103,169.892,48.659,159.338
C04443=1023.025,264.269,-128.153,169.899,48.653,159.338
C04444=1023.032,264.517,-128.182,169.904,48.650,159.338
C04445=1023.039,264.765,-128.212,169.908,48.647,159.338
C04446=1023.045,265.013,-128.241,169.912,48.643,159.337
C04447=1023.051,265.262,-128.270,169.916,48.641,159.337
C04448=1023.059,265.510,-128.300,169.920,48.637,159.337
C04449=1023.065,265.758,-128.329,169.925,48.634,159.337
C04450=1023.071,266.006,-128.360,169.929,48.631,159.337
C04451=1023.077,266.255,-128.389,169.933,48.627,159.337
C04452=1023.084,266.503,-128.418,169.937,48.624,159.337
C04453=1023.090,266.750,-128.448,169.941,48.621,159.337
C04454=1023.096,266.999,-128.478,169.946,48.618,159.337
C04455=1023.103,267.247,-128.508,169.950,48.615,159.337
C04456=1023.109,267.495,-128.537,169.954,48.612,159.337
C04457=1023.116,267.744,-128.567,169.958,48.608,159.336
C04458=1023.122,267.991,-128.597,169.962,48.606,159.336
C04459=1023.128,268.239,-128.626,169.967,48.602,159.336
C04460=1023.135,268.488,-128.657,169.972,48.599,159.336
C04461=1023.141,268.736,-128.686,169.976,48.596,159.336
C04462=1023.148,268.984,-128.716,169.980,48.593,159.336
C04463=1023.155,269.232,-128.746,169.984,48.590,159.336
C04464=1023.160,269.480,-128.775,169.988,48.586,159.336
C04465=1023.167,269.728,-128.805,169.993,48.584,159.336
C04466=1023.174,269.976,-128.835,169.997,48.581,159.336
C04467=1023.180,270.225,-128.865,170.001,48.577,159.336
C04468=1023.187,270.472,-128.895,170.006,48.575,159.336
C04469=1023.193,270.721,-128.926,170.010,48.572,159.336
C04470=1023.200,270.968,-128.955,170.014,48.568,159.336
C04471=1023.205,271.217,-128.985,170.018,48.566,159.336
C04472=1023.212,271.465,-129.015,170.023,48.563,159.336
C04473=1023.218,271.713,-129.046,170.027,48.560,159.336
C04474=1023.225,271.961,-129.076,170.032,48.556,159.336
C04475=1023.231,272.209,-129.106,170.036,48.553,159.336
C04476=1023.238,272.457,-129.136,170.041,48.550,159.336
C04477=1023.244,272.706,-129.166,170.045,48.548,159.336
C04478=1023.251,272.954,-129.196,170.049,48.544,159.335
C04479=1023.257,273.202,-129.226,170.054,48.541,159.335
C04480=1023.264,273.450,-129.256,170.058,48.539,159.335
C04481=1023.270,273.698,-129.287,170.062,48.536,159.335
C04482=1023.277,273.946,-129.317,170.067,48.533,159.335
C04483=1023.283,274.194,-129.347,170.071,48.530,159.335
C04484=1023.290,274.442,-129.377,170.075,48.527,159.335
C04485=1023.296,274.690,-129.408,170.079,48.524,159.335
C04486=1023.303,274.938,-129.438,170.084,48.521,159.335
C04487=1023.309,275.186,-129.468,170.089,48.518,159.335
C04488=1023.315,275.434,-129.499,170.094,48.515,159.335
C04489=1023.322,275.682,-129.529,170.098,48.512,159.335
C04490=1023.328,275.930,-129.559,170.102,48.510,159.335
C04491=1023.335,276.178,-129.589,170.107,48.507,159.335
C04492=1023.341,276.426,-129.620,170.111,48.504,159.335
C04493=1023.348,276.675,-129.650,170.115,48.501,159.335
C04494=1023.354,276.922,-129.681,170.120,48.498,159.335
C04495=1023.361,277.170,-129.712,170.124,48.496,159.335
C04496=1023.366,277.382,-129.737,170.129,48.493,159.335
C04497=1023.372,277.593,-129.763,170.132,48.490,159.335
C04498=1023.378,277.804,-129.790,170.136,48.488,159.335
C04499=1023.382,278.016,-129.816,170.139,48.486,159.335
C04500=1023.388,278.227,-129.842,170.144,48.484,159.335
C04501=1023.394,278.439,-129.868,170.147,48.481,159.335
C04502=1023.399,278.650,-129.894,170.150,48.479,159.335
C04503=1023.405,278.861,-129.920,170.155,48.477,159.336
C04504=1023.411,279.109,-129.951,170.159,48.474,159.336
C04505=1023.418,279.358,-129.982,170.164,48.471,159.336
C04506=1023.424,279.605,-130.013,170.168,48.468,159.336
C04507=1023.430,279.853,-130.043,170.173,48.465,159.336
C04508=1023.437,280.101,-130.075,170.177,48.463,159.336
C04509=1023.444,280.349,-130.105,170.182,48.460,159.336
C04510=1023.450,280.597,-130.135,170.186,48.458,159.336
C04511=1023.457,280.845,-130.167,170.190,48.455,159.336
C04512=1023.463,281.093,-130.197,170.195,48.452,159.336
C04513=1023.469,281.341,-130.228,170.200,48.450,159.336
C04514=1023.476,281.589,-130.259,170.205,48.447,159.336
C04515=1023.483,281.837,-130.290,170.209,48.444,159.336
C04516=1023.489,282.085,-130.320,170.214,48.441,159.336
C04517=1023.496,282.333,-130.352,170.218,48.439,159.336
C04518=1023.502,282.581,-130.382,170.223,48.436,159.336
C04519=1023.509,282.829,-130.414,170.227,48.433,159.336
C04520=1023.515,283.077,-130.444,170.231,48.431,159.336
C04521=1023.522,283.325,-130.475,170.236,48.428,159.336
C04522=1023.529,283.573,-130.506,170.240,48.426,159.336
C04523=1023.535,283.821,-130.537,170.246,48.423,159.336
C04524=1023.541,284.069,-130.568,170.251,48.420,159.337
C04525=1023.548,284.317,-130.599,170.255,48.418,159.337
C04526=1023.555,284.564,-130.630,170.259,48.415,159.337
C04527=1023.562,284.813,-130.661,170.264,48.413,159.337
C04528=1023.568,285.061,-130.692,170.268,48.410,159.337
C04529=1023.575,285.309,-130.723,170.273,48.408,159.337
C04530=1023.581,285.557,-130.754,170.277,48.405,159.337
C04531=1023.588,285.804,-130.785,170.283,48.403,159.337
C04532=1023.594,286.052,-130.817,170.288,48.400,159.337
C04533=1023.601,286.300,-130.848,170.292,48.398,159.337
C04534=1023.608,286.549,-130.879,170.297,48.395,159.337
C04535=1023.614,286.797,-130.910,170.301,48.393,159.338
C04536=1023.621,287.045,-130.942,170.306,48.390,159.338
C04537=1023.627,287.292,-130.973,170.310,48.388,159.338
C04538=1023.634,287.540,-131.004,170.315,48.385,159.338
C04539=1023.641,287.788,-131.036,170.319,48.383,159.338
C04540=1023.647,288.035,-131.067,170.325,48.380,159.338
C04541=1023.654,288.283,-131.098,170.330,48.378,159.338
C04542=1023.660,288.532,-131.131,170.334,48.375,159.338
C04543=1023.667,288.779,-131.162,170.339,48.373,159.338
C04544=1023.673,289.027,-131.193,170.343,48.370,159.339
C04545=1023.680,289.275,-131.225,170.348,48.368,159.339
C04546=1023.687,289.523,-131.256,170.352,48.366,159.339
C04547=1023.694,289.771,-131.288,170.357,48.363,159.339
C04548=1023.700,290.019,-131.319,170.363,48.361,159.339
C04549=1023.706,290.267,-131.351,170.367,48.358,159.339
C04550=1023.712,290.514,-131.382,170.372,48.356,159.339
C04551=1023.719,290.762,-131.414,170.377,48.354,159.340
C04552=1023.726,291.010,-131.445,170.381,48.352,159.340
C04553=1023.733,291.258,-131.477,170.386,48.349,159.340
C04554=1023.739,291.506,-131.508,170.390,48.347,159.340
C04555=1023.746,291.754,-131.539,170.396,48.344,159.340
C04556=1023.752,291.971,-131.568,170.400,48.342,159.340
C04557=1023.758,292.189,-131.596,170.404,48.340,159.341
C04558=1023.764,292.407,-131.623,170.408,48.339,159.341
C04559=1023.769,292.624,-131.651,170.413,48.336,159.341
C04560=1023.775,292.841,-131.680,170.417,48.335,159.341
C04561=1023.781,293.059,-131.707,170.421,48.332,159.341
C04562=1023.787,293.277,-131.735,170.425,48.331,159.341
C04563=1023.793,293.493,-131.763,170.430,48.328,159.341
C04564=1023.799,293.741,-131.795,170.434,48.326,159.342
C04565=1023.805,293.989,-131.827,170.439,48.324,159.342
C04566=1023.812,294.237,-131.859,170.444,48.322,159.342
C04567=1023.818,294.485,-131.891,170.448,48.320,159.342
C04568=1023.825,294.733,-131.924,170.453,48.318,159.342
C04569=1023.832,294.981,-131.955,170.458,48.316,159.343
C04570=1023.838,295.229,-131.988,170.463,48.313,159.343
C04571=1023.844,295.477,-132.020,170.468,48.311,159.343
C04572=1023.851,295.724,-132.052,170.473,48.309,159.343
C04573=1023.858,295.972,-132.085,170.478,48.307,159.343
C04574=1023.864,296.220,-132.117,170.483,48.305,159.344
C04575=1023.871,296.467,-132.149,170.487,48.303,159.344
C04576=1023.877,296.716,-132.181,170.492,48.301,159.344
C04577=1023.884,296.963,-132.213,170.497,48.299,159.344
C04578=1023.890,297.210,-132.246,170.502,48.297,159.344
C04579=1023.897,297.459,-132.278,170.507,48.294,159.345
C04580=1023.903,297.707,-132.311,170.512,48.293,159.345
C04581=1023.910,297.954,-132.343,170.517,48.291,159.345
C04582=1023.916,298.202,-132.375,170.522,48.288,159.345
C04583=1023.923,298.450,-132.408,170.526,48.286,159.346
C04584=1023.929,298.697,-132.440,170.531,48.284,159.346
C04585=1023.937,298.945,-132.473,170.536,48.283,159.346
C04586=1023.943,299.194,-132.505,170.542,48.280,159.346
C04587=1023.950,299.441,-132.537,170.547,48.278,159.347
C04588=1023.956,299.688,-132.570,170.552,48.277,159.347
C04589=1023.962,299.936,-132.603,170.556,48.274,159.347
C04590=1023.970,300.184,-132.635,170.561,48.272,159.347
C04591=1023.976,300.432,-132.667,170.566,48.270,159.348
C04592=1023.982,300.680,-132.700,170.572,48.268,159.348
C04593=1023.989,300.927,-132.732,170.577,48.266,159.348
C04594=1023.996,301.175,-132.765,170.581,48.264,159.348
C04595=1024.003,301.423,-132.797,170.586,48.263,159.349
C04596=1024.009,301.670,-132.830,170.591,48.260,159.349
C04597=1024.016,301.919,-132.863,170.597,48.259,159.349
C04598=1024.023,302.166,-132.895,170.602,48.257,159.350
C04599=1024.030,302.413,-132.928,170.606,48.254,159.350
C04600=1024.037,302.662,-132.961,170.611,48.253,159.350
C04601=1024.044,302.909,-132.993,170.616,48.251,159.350
C04602=1024.050,303.157,-133.026,170.622,48.249,159.351
C04603=1024.057,303.405,-133.059,170.627,48.247,159.351
C04604=1024.064,303.652,-133.091,170.632,48.245,159.351
C04605=1024.070,303.900,-133.124,170.637,48.243,159.351
C04606=1024.078,304.148,-133.156,170.643,48.241,159.352
C04607=1024.084,304.395,-133.189,170.647,48.239,159.352
C04608=1024.091,304.644,-133.222,170.652,48.238,159.352
C04609=1024.098,304.891,-133.254,170.657,48.236,159.353
C04610=1024.105,305.139,-133.288,170.663,48.234,159.353
C04611=1024.111,305.386,-133.321,170.668,48.232,159.353
C04612=1024.118,305.633,-133.353,170.673,48.230,159.354
C04613=1024.125,305.882,-133.386,170.678,48.228,159.354
C04614=1024.132,306.129,-133.419,170.684,48.226,159.354
C04615=1024.139,306.377,-133.452,170.689,48.225,159.355
C04616=1024.146,306.603,-133.482,170.693,48.223,159.355
C04617=1024.152,306.829,-133.511,170.697,48.221,159.355
C04618=1024.158,307.055,-133.542,170.702,48.219,159.355
C04619=1024.164,307.281,-133.573,170.707,48.218,159.356
C04620=1024.171,307.508,-133.602,170.712,48.216,159.356
C04621=1024.177,307.733,-133.632,170.717,48.215,159.356
C04622=1024.184,307.960,-133.662,170.722,48.213,159.356
C04623=1024.190,308.186,-133.693,170.726,48.211,159.357
C04624=1024.197,308.434,-133.726,170.732,48.210,159.357
C04625=1024.204,308.681,-133.758,170.737,48.208,159.357
C04626=1024.211,308.929,-133.792,170.742,48.206,159.358
C04627=1024.218,309.178,-133.825,170.748,48.204,159.358
C04628=1024.225,309.424,-133.858,170.753,48.203,159.359
C04629=1024.232,309.672,-133.891,170.758,48.201,159.359
C04630=1024.239,309.919,-133.924,170.764,48.199,159.359
C04631=1024.246,310.167,-133.957,170.769,48.197,159.359
C04632=1024.254,310.415,-133.990,170.774,48.196,159.360
C04633=1024.260,310.663,-134.023,170.779,48.194,159.360
C04634=1024.267,310.910,-134.057,170.785,48.193,159.361
C04635=1024.273,311.158,-134.091,170.790,48.191,159.361
C04636=1024.280,311.405,-134.125,170.795,48.190,159.361
C04637=1024.286,311.653,-134.158,170.800,48.188,159.362
C04638=1024.293,311.901,-134.192,170.806,48.186,159.362
C04639=1024.300,312.149,-134.226,170.811,48.185,159.363
C04640=1024.307,312.396,-134.259,170.816,48.183,159.363
C04641=1024.314,312.643,-134.293,170.821,48.182,159.363
C04642=1024.320,312.891,-134.327,170.827,48.180,159.364
C04643=1024.327,313.139,-134.360,170.832,48.179,159.364
C04644=1024.334,313.386,-134.394,170.837,48.178,159.365
C04645=1024.340,313.633,-134.428,170.843,48.176,159.365
C04646=1024.347,313.881,-134.462,170.849,48.174,159.365
C04647=1024.354,314.129,-134.496,170.854,48.173,159.366
C04648=1024.361,314.377,-134.530,170.859,48.171,159.366
C04649=1024.367,314.624,-134.564,170.864,48.171,159.367
C04650=1024.374,314.872,-134.598,170.870,48.169,159.367
C04651=1024.382,315.119,-134.631,170.875,48.167,159.367
C04652=1024.387,315.367,-134.665,170.880,48.166,159.368
C04653=1024.395,315.614,-134.699,170.886,48.165,159.368
C04654=1024.402,315.862,-134.733,170.892,48.163,159.369
C04655=1024.409,316.109,-134.768,170.897,48.162,159.369
C04656=1024.416,316.357,-134.802,170.903,48.160,159.370
C04657=1024.422,316.604,-134.836,170.908,48.159,159.370
C04658=1024.430,316.852,-134.869,170.913,48.157,159.371
C04659=1024.436,317.100,-134.904,170.919,48.156,159.371
C04660=1024.443,317.347,-134.938,170.924,48.155,159.372
C04661=1024.450,317.595,-134.971,170.929,48.153,159.372
C04662=1024.457,317.842,-135.007,170.936,48.152,159.372
C04663=1024.464,318.089,-135.040,170.941,48.151,159.373
C04664=1024.471,318.337,-135.074,170.946,48.149,159.373
C04665=1024.478,318.585,-135.108,170.952,48.148,159.374
C04666=1024.485,318.832,-135.143,170.957,48.146,159.374
C04667=1024.492,319.080,-135.177,170.963,48.146,159.375
C04668=1024.499,319.327,-135.210,170.969,48.144,159.375
C04669=1024.506,319.575,-135.246,170.974,48.143,159.376
C04670=1024.513,319.823,-135.279,170.979,48.141,159.376
C04671=1024.521,320.070,-135.313,170.985,48.140,159.377
C04672=1024.527,320.318,-135.348,170.990,48.139,159.377
C04673=1024.535,320.565,-135.382,170.997,48.138,159.378
C04674=1024.542,320.813,-135.416,171.002,48.136,159.378
C04675=1024.549,321.060,-135.451,171.007,48.135,159.379
C04676=1024.555,321.289,-135.482,171.012,48.134,159.379
C04677=1024.562,321.518,-135.514,171.018,48.133,159.380
C04678=1024.569,321.747,-135.545,171.023,48.131,159.380
C04679=1024.575,321.975,-135.578,171.028,48.131,159.380
C04680=1024.582,322.204,-135.610,171.033,48.130,159.381
C04681=1024.588,322.432,-135.641,171.038,48.128,159.381
C04682=1024.595,322.660,-135.673,171.044,48.127,159.382
C04683=1024.601,322.890,-135.705,171.049,48.126,159.382
C04684=1024.609,323.137,-135.740,171.055,48.125,159.383
C04685=1024.616,323.385,-135.774,171.061,48.124,159.383
C04686=1024.623,323.632,-135.809,171.067,48.122,159.384
C04687=1024.630,323.880,-135.843,171.072,48.121,159.384
C04688=1024.638,324.127,-135.878,171.078,48.120,159.385
C04689=1024.645,324.375,-135.913,171.084,48.119,159.386
C04690=1024.652,324.622,-135.947,171.090,48.117,159.386
C04691=1024.659,324.869,-135.981,171.095,48.116,159.387
C04692=1024.666,325.117,-136.016,171.101,48.115,159.387
C04693=1024.674,325.365,-136.050,171.107,48.114,159.388
C04694=1024.681,325.612,-136.085,171.113,48.113,159.388
C04695=1024.688,325.860,-136.120,171.118,48.112,159.389
C04696=1024.696,326.107,-136.155,171.124,48.111,159.389
C04697=1024.703,326.355,-136.189,171.130,48.110,159.390
C04698=1024.710,326.602,-136.224,171.135,48.109,159.390
C04699=1024.718,326.850,-136.259,171.142,48.108,159.391
C04700=1024.725,327.097,-136.294,171.147,48.107,159.392
C04701=1024.733,327.345,-136.329,171.153,48.106,159.392
C04702=1024.739,327.592,-136.364,171.159,48.105,159.393
C04703=1024.746,327.839,-136.399,171.165,48.104,159.393
C04704=1024.753,328.087,-136.434,171.171,48.103,159.394
C04705=1024.761,328.334,-136.469,171.177,48.102,159.394
C04706=1024.768,328.582,-136.504,171.182,48.101,159.395
C04707=1024.775,328.829,-136.540,171.189,48.100,159.396
C04708=1024.782,329.077,-136.575,171.194,48.099,159.396
C04709=1024.789,329.324,-136.610,171.201,48.098,159.397
C04710=1024.797,329.571,-136.645,171.206,48.097,159.398
C04711=1024.804,329.819,-136.681,171.212,48.096,159.398
C04712=1024.811,330.066,-136.716,171.218,48.095,159.399
C04713=1024.818,330.313,-136.752,171.224,48.094,159.399
C04714=1024.825,330.561,-136.787,171.230,48.094,159.400
C04715=1024.833,330.808,-136.822,171.236,48.093,159.401
C04716=1024.840,331.055,-136.857,171.242,48.092,159.401
C04717=1024.847,331.303,-136.893,171.248,48.091,159.402
C04718=1024.854,331.551,-136.928,171.254,48.090,159.403
C04719=1024.862,331.798,-136.964,171.260,48.089,159.403
C04720=1024.869,332.045,-136.999,171.265,48.088,159.404
C04721=1024.877,332.292,-137.035,171.272,48.088,159.405
C04722=1024.884,332.540,-137.070,171.277,48.087,159.405
C04723=1024.891,332.787,-137.106,171.284,48.086,159.406
C04724=1024.898,333.035,-137.141,171.291,48.085,159.406
C04725=1024.906,333.282,-137.176,171.296,48.084,159.407
C04726=1024.913,333.529,-137.212,171.303,48.084,159.408
C04727=1024.921,333.777,-137.248,171.308,48.083,159.408
C04728=1024.928,334.024,-137.284,171.315,48.082,159.409
C04729=1024.935,334.271,-137.320,171.320,48.082,159.410
C04730=1024.942,334.518,-137.356,171.327,48.081,159.411
C04731=1024.950,334.766,-137.391,171.332,48.080,159.411
C04732=1024.957,335.013,-137.427,171.339,48.080,159.412
C04733=1024.964,335.261,-137.464,171.345,48.079,159.413
C04734=1024.971,335.507,-137.500,171.351,48.078,159.413
C04735=1024.978,335.756,-137.535,171.358,48.078,159.414
C04736=1024.985,335.981,-137.568,171.363,48.077,159.415
C04737=1024.992,336.209,-137.601,171.369,48.077,159.415
C04738=1024.999,336.435,-137.634,171.374,48.076,159.416
C04739=1025.005,336.661,-137.666,171.380,48.075,159.417
C04740=1025.012,336.887,-137.700,171.385,48.075,159.417
C04741=1025.020,337.114,-137.733,171.392,48.074,159.418
C04742=1025.025,337.341,-137.766,171.397,48.074,159.419
C04743=1025.032,337.567,-137.799,171.403,48.073,159.419
C04744=1025.040,337.814,-137.835,171.408,48.073,159.420
C04745=1025.047,338.061,-137.872,171.415,48.072,159.421
C04746=1025.055,338.309,-137.908,171.422,48.071,159.422
C04747=1025.062,338.556,-137.944,171.427,48.071,159.422
C04748=1025.070,338.803,-137.980,171.434,48.070,159.423
C04749=1025.077,339.050,-138.016,171.441,48.070,159.424
C04750=1025.085,339.298,-138.052,171.446,48.069,159.424
C04751=1025.092,339.545,-138.088,171.453,48.069,159.425
C04752=1025.100,339.792,-138.124,171.460,48.068,159.426
C04753=1025.107,340.040,-138.161,171.465,48.068,159.427
C04754=1025.115,340.287,-138.198,171.472,48.067,159.428
C04755=1025.122,340.533,-138.234,171.479,48.067,159.428
C04756=1025.130,340.781,-138.270,171.484,48.067,159.429
C04757=1025.137,341.029,-138.307,171.491,48.066,159.430
C04758=1025.145,341.275,-138.344,171.498,48.065,159.431
C04759=1025.152,341.523,-138.380,171.504,48.065,159.431
C04760=1025.159,341.771,-138.417,171.510,48.065,159.432
C04761=1025.166,342.017,-138.453,171.517,48.064,159.433
C04762=1025.174,342.264,-138.490,171.523,48.064,159.434
C04763=1025.181,342.511,-138.527,171.529,48.063,159.435
C04764=1025.189,342.759,-138.563,171.536,48.063,159.436
C04765=1025.197,343.006,-138.600,171.543,48.063,159.436
C04766=1025.204,343.253,-138.637,171.549,48.063,159.437
C04767=1025.212,343.501,-138.673,171.555,48.062,159.438
C04768=1025.220,343.748,-138.710,171.562,48.062,159.439
C04769=1025.227,343.995,-138.748,171.568,48.062,159.440
C04770=1025.235,344.242,-138.784,171.575,48.061,159.440
C04771=1025.242,344.489,-138.822,171.582,48.061,159.441
C04772=1025.250,344.737,-138.858,171.589,48.061,159.442
C04773=1025.257,344.984,-138.895,171.594,48.060,159.443
C04774=1025.265,345.231,-138.932,171.601,48.060,159.444
C04775=1025.272,345.478,-138.968,171.608,48.060,159.445
C04776=1025.280,345.725,-139.006,171.615,48.059,159.446
C04777=1025.288,345.972,-139.043,171.622,48.059,159.447
C04778=1025.295,346.219,-139.080,171.627,48.059,159.447
C04779=1025.303,346.467,-139.117,171.634,48.059,159.448
C04780=1025.311,346.714,-139.154,171.641,48.059,159.449
C04781=1025.318,346.961,-139.191,171.648,48.058,159.450
C04782=1025.326,347.208,-139.228,171.654,48.058,159.451
C04783=1025.333,347.455,-139.266,171.661,48.058,159.452
C04784=1025.341,347.702,-139.303,171.668,48.058,159.453
C04785=1025.349,347.949,-139.340,171.675,48.058,159.454
C04786=1025.357,348.196,-139.377,171.681,48.057,159.454
C04787=1025.364,348.443,-139.415,171.688,48.058,159.455
C04788=1025.372,348.690,-139.452,171.694,48.058,159.456
C04789=1025.379,348.937,-139.489,171.701,48.057,159.457
C04790=1025.387,349.184,-139.527,171.708,48.057,159.458
C04791=1025.395,349.432,-139.564,171.715,48.057,159.459
C04792=1025.402,349.679,-139.602,171.722,48.057,159.460
C04793=1025.410,349.926,-139.639,171.729,48.057,159.461
C04794=1025.418,350.172,-139.677,171.735,48.057,159.462
C04795=1025.425,350.420,-139.714,171.742,48.057,159.463
C04796=1025.432,350.645,-139.748,171.749,48.057,159.464
C04797=1025.439,350.870,-139.783,171.755,48.057,159.465
C04798=1025.446,351.094,-139.818,171.761,48.057,159.465
C04799=1025.453,351.320,-139.852,171.767,48.057,159.466
C04800=1025.461,351.544,-139.886,171.773,48.057,159.467
C04801=1025.468,351.770,-139.920,171.779,48.057,159.468
C04802=1025.475,351.994,-139.954,171.786,48.057,159.469
C04803=1025.481,352.219,-139.989,171.792,48.057,159.470
C04804=1025.490,352.466,-140.027,171.799,48.057,159.471
C04805=1025.497,352.713,-140.065,171.806,48.057,159.472
C04806=1025.505,352.960,-140.102,171.813,48.057,159.473
C04807=1025.514,353.207,-140.140,171.820,48.058,159.474
C04808=1025.521,353.454,-140.178,171.827,48.058,159.475
C04809=1025.529,353.701,-140.216,171.834,48.058,159.476
C04810=1025.536,353.948,-140.254,171.841,48.058,159.477
C04811=1025.545,354.195,-140.292,171.848,48.058,159.478
C04812=1025.552,354.442,-140.330,171.855,48.058,159.479
C04813=1025.560,354.689,-140.368,171.862,48.058,159.480
C04814=1025.568,354.936,-140.406,171.869,48.058,159.481
C04815=1025.576,355.183,-140.443,171.877,48.058,159.482
C04816=1025.584,355.430,-140.482,171.884,48.059,159.483
C04817=1025.592,355.677,-140.520,171.891,48.059,159.484
C04818=1025.600,355.924,-140.559,171.898,48.059,159.485
C04819=1025.607,356.170,-140.597,171.905,48.059,159.486
C04820=1025.615,356.418,-140.635,171.912,48.059,159.487
C04821=1025.623,356.665,-140.673,171.919,48.059,159.488
C04822=1025.631,356.912,-140.712,171.927,48.060,159.489
C04823=1025.639,357.159,-140.750,171.934,48.060,159.490
C04824=1025.647,357.405,-140.788,171.941,48.061,159.491
C04825=1025.656,357.653,-140.827,171.948,48.061,159.492
C04826=1025.663,357.899,-140.865,171.955,48.061,159.493
C04827=1025.671,358.146,-140.903,171.962,48.061,159.495
C04828=1025.679,358.393,-140.942,171.969,48.061,159.496
C04829=1025.687,358.640,-140.980,171.977,48.062,159.497
C04830=1025.695,358.887,-141.019,171.984,48.062,159.498
C04831=1025.704,359.134,-141.058,171.991,48.063,159.499
C04832=1025.711,359.380,-141.097,171.998,48.063,159.500
C04833=1025.719,359.628,-141.135,172.005,48.063,159.501
C04834=1025.727,359.875,-141.174,172.013,48.064,159.502
C04835=1025.735,360.121,-141.212,172.021,48.064,159.503
C04836=1025.743,360.368,-141.251,172.028,48.064,159.505
C04837=1025.752,360.615,-141.290,172.036,48.065,159.506
C04838=1025.760,360.862,-141.329,172.043,48.066,159.507
C04839=1025.768,361.108,-141.367,172.050,48.066,159.508
C04840=1025.775,361.356,-141.407,172.057,48.066,159.509
C04841=1025.784,361.602,-141.446,172.065,48.067,159.510
C04842=1025.792,361.849,-141.485,172.072,48.068,159.512
C04843=1025.800,362.096,-141.524,172.079,48.068,159.513
C04844=1025.807,362.342,-141.564,172.088,48.069,159.514
C04845=1025.815,362.590,-141.602,172.095,48.069,159.515
C04846=1025.824,362.836,-141.641,172.103,48.070,159.516
C04847=1025.832,363.083,-141.680,172.110,48.070,159.518
C04848=1025.840,363.330,-141.719,172.117,48.071,159.519
C04849=1025.848,363.577,-141.759,172.126,48.071,159.520
C04850=1025.856,363.823,-141.798,172.133,48.072,159.521
C04851=1025.864,364.070,-141.837,172.140,48.073,159.522
C04852=1025.873,364.317,-141.876,172.148,48.073,159.524
C04853=1025.880,364.563,-141.916,172.155,48.074,159.525
C04854=1025.889,364.810,-141.955,172.163,48.074,159.526
C04855=1025.897,365.057,-141.994,172.171,48.075,159.527
C04856=1025.905,365.285,-142.031,172.178,48.076,159.528
C04857=1025.913,365.513,-142.067,172.184,48.076,159.530
C04858=1025.920,365.742,-142.103,172.192,48.077,159.531
C04859=1025.928,365.970,-142.140,172.199,48.078,159.532
C04860=1025.935,366.198,-142.177,172.206,48.078,159.533
C04861=1025.943,366.427,-142.214,172.214,48.078,159.534
C04862=1025.951,366.655,-142.250,172.220,48.079,159.535
C04863=1025.959,366.884,-142.286,172.227,48.080,159.536
C04864=1025.967,367.130,-142.326,172.236,48.081,159.538
C04865=1025.976,367.376,-142.366,172.243,48.081,159.539
C04866=1025.984,367.623,-142.406,172.251,48.082,159.540
C04867=1025.992,367.870,-142.445,172.259,48.083,159.542
C04868=1026.000,368.116,-142.484,172.267,48.084,159.543
C04869=1026.009,368.363,-142.524,172.274,48.085,159.544
C04870=1026.017,368.610,-142.564,172.283,48.085,159.545
C04871=1026.026,368.856,-142.604,172.291,48.086,159.547
C04872=1026.034,369.103,-142.644,172.298,48.087,159.548
C04873=1026.042,369.350,-142.683,172.307,48.088,159.549
C04874=1026.050,369.596,-142.724,172.314,48.088,159.551
C04875=1026.059,369.843,-142.763,172.323,48.089,159.552
C04876=1026.067,370.090,-142.804,172.330,48.091,159.554
C04877=1026.076,370.336,-142.843,172.338,48.091,159.555
C04878=1026.084,370.583,-142.884,172.346,48.092,159.556
C04879=1026.092,370.829,-142.925,172.354,48.093,159.558
C04880=1026.101,371.076,-142.964,172.363,48.094,159.559
C04881=1026.109,371.323,-143.005,172.370,48.095,159.560
C04882=1026.117,371.569,-143.044,172.378,48.096,159.562
C04883=1026.126,371.816,-143.085,172.387,48.097,159.563
C04884=1026.135,372.062,-143.125,172.394,48.098,159.564
C04885=1026.143,372.308,-143.166,172.403,48.099,159.566
C04886=1026.151,372.556,-143.206,172.411,48.100,159.567
C04887=1026.160,372.802,-143.246,172.419,48.101,159.569
C04888=1026.168,373.049,-143.287,172.427,48.102,159.570
C04889=1026.177,373.295,-143.327,172.436,48.103,159.572
C04890=1026.185,373.541,-143.368,172.443,48.104,159.573
C04891=1026.194,373.788,-143.409,172.452,48.105,159.574
C04892=1026.203,374.034,-143.449,172.460,48.107,159.576
C04893=1026.211,374.282,-143.489,172.469,48.107,159.577
C04894=1026.220,374.528,-143.529,172.476,48.109,159.579
C04895=1026.228,374.775,-143.570,172.485,48.109,159.580
C04896=1026.237,375.020,-143.611,172.494,48.110,159.581
C04897=1026.246,375.267,-143.652,172.501,48.112,159.583
C04898=1026.255,375.514,-143.693,172.510,48.113,159.585
C04899=1026.263,375.760,-143.733,172.518,48.114,159.586
C04900=1026.272,376.007,-143.774,172.527,48.115,159.587
C04901=1026.281,376.253,-143.814,172.535,48.116,159.589
C04902=1026.289,376.500,-143.855,172.544,48.118,159.590
C04903=1026.298,376.746,-143.897,172.552,48.119,159.592
C04904=1026.307,376.992,-143.937,172.560,48.120,159.593
C04905=1026.316,377.239,-143.978,172.569,48.121,159.595
C04906=1026.325,377.486,-144.020,172.578,48.122,159.596
C04907=1026.333,377.732,-144.060,172.586,48.124,159.598
C04908=1026.342,377.978,-144.102,172.594,48.125,159.599
C04909=1026.350,378.225,-144.143,172.603,48.126,159.601
C04910=1026.359,378.471,-144.184,172.611,48.128,159.603
C04911=1026.367,378.718,-144.225,172.620,48.129,159.604
C04912=1026.376,378.964,-144.267,172.629,48.131,159.606
C04913=1026.385,379.210,-144.308,172.637,48.132,159.607
C04914=1026.394,379.457,-144.349,172.646,48.133,159.609
C04915=1026.403,379.703,-144.391,172.655,48.135,159.610
C04916=1026.412,379.942,-144.431,172.663,48.136,159.612
C04917=1026.420,380.181,-144.471,172.672,48.137,159.613
C04918=1026.429,380.420,-144.512,172.681,48.139,159.615
C04919=1026.437,380.658,-144.551,172.688,48.140,159.616
C04920=1026.446,380.897,-144.592,172.698,48.141,159.618
C04921=1026.453,381.136,-144.632,172.706,48.143,159.620
C04922=1026.462,381.375,-144.673,172.714,48.144,159.621
C04923=1026.471,381.614,-144.713,172.722,48.146,159.623
C04924=1026.480,381.860,-144.755,172.731,48.147,159.624
C04925=1026.489,382.106,-144.796,172.740,48.149,159.626
C04926=1026.498,382.352,-144.838,172.749,48.150,159.628
C04927=1026.507,382.599,-144.880,172.758,48.152,159.629
C04928=1026.516,382.845,-144.921,172.768,48.153,159.631
C04929=1026.525,383.092,-144.963,172.777,48.154,159.633
C04930=1026.534,383.338,-145.005,172.785,48.156,159.634
C04931=1026.543,383.584,-145.047,172.794,48.158,159.636
C04932=1026.552,383.831,-145.088,172.803,48.160,159.638
C04933=1026.561,384.076,-145.131,172.812,48.161,159.639
C04934=1026.571,384.323,-145.173,172.821,48.163,159.641
C04935=1026.580,384.570,-145.214,172.830,48.164,159.643
C04936=1026.589,384.816,-145.257,172.840,48.166,159.645
C04937=1026.598,385.062,-145.299,172.849,48.168,159.646
C04938=1026.607,385.308,-145.340,172.858,48.169,159.648
C04939=1026.616,385.554,-145.383,172.867,48.171,159.650
C04940=1026.626,385.801,-145.425,172.876,48.172,159.651
C04941=1026.635,386.047,-145.467,172.885,48.174,159.653
C04942=1026.644,386.293,-145.509,172.894,48.176,159.655
C04943=1026.653,386.539,-145.551,172.904,48.178,159.657
C04944=1026.663,386.786,-145.594,172.913,48.179,159.658
C04945=1026.672,387.032,-145.636,172.922,48.181,159.660
C04946=1026.681,387.277,-145.678,172.931,48.183,159.662
C04947=1026.689,387.524,-145.721,172.941,48.185,159.664
C04948=1026.699,387.771,-145.763,172.950,48.187,159.666
C04949=1026.708,388.016,-145.806,172.960,48.189,159.668
C04950=1026.718,388.262,-145.848,172.970,48.190,159.669
C04951=1026.727,388.509,-145.891,172.979,48.192,159.671
C04952=1026.736,388.755,-145.934,172.988,48.194,159.673
C04953=1026.746,389.001,-145.977,172.998,48.196,159.675
C04954=1026.755,389.247,-146.019,173.007,48.198,159.677
C04955=1026.764,389.492,-146.062,173.016,48.199,159.678
C04956=1026.773,389.739,-146.105,173.026,48.201,159.680
C04957=1026.783,389.985,-146.148,173.036,48.203,159.682
C04958=1026.792,390.231,-146.190,173.045,48.205,159.684
C04959=1026.801,390.477,-146.234,173.055,48.208,159.686
C04960=1026.811,390.723,-146.277,173.064,48.210,159.688
C04961=1026.820,390.969,-146.319,173.074,48.212,159.690
C04962=1026.830,391.215,-146.364,173.084,48.213,159.692
C04963=1026.839,391.461,-146.406,173.094,48.215,159.694
C04964=1026.848,391.708,-146.449,173.103,48.217,159.695
C04965=1026.858,391.954,-146.493,173.113,48.220,159.697
C04966=1026.867,392.199,-146.535,173.123,48.222,159.699
C04967=1026.877,392.445,-146.579,173.133,48.224,159.701
C04968=1026.886,392.691,-146.622,173.142,48.226,159.703
C04969=1026.896,392.937,-146.665,173.153,48.228,159.705
C04970=1026.905,393.184,-146.709,173.162,48.230,159.707
C04971=1026.915,393.430,-146.752,173.172,48.232,159.709
C04972=1026.924,393.675,-146.796,173.182,48.234,159.711
C04973=1026.934,393.921,-146.839,173.192,48.237,159.713
C04974=1026.943,394.168,-146.883,173.201,48.239,159.715
C04975=1026.953,394.413,-146.926,173.212,48.241,159.717
C04976=1026.964,394.681,-146.974,173.223,48.243,159.719
C04977=1026.973,394.949,-147.022,173.234,48.246,159.722
C04978=1026.984,395.216,-147.069,173.245,48.248,159.724
C04979=1026.995,395.484,-147.117,173.255,48.250,159.726
C04980=1027.004,395.731,-147.161,173.266,48.253,159.728
C04981=1027.015,395.976,-147.205,173.276,48.255,159.730
C04982=1027.023,396.222,-147.248,173.286,48.258,159.732
C04983=1027.033,396.468,-147.292,173.296,48.260,159.734
C04984=1027.043,396.714,-147.336,173.307,48.262,159.736
C04985=1027.053,396.960,-147.380,173.316,48.264,159.738
C04986=1027.063,397.205,-147.424,173.327,48.266,159.740
C04987=1027.073,397.451,-147.468,173.337,48.269,159.742
C04988=1027.082,397.697,-147.512,173.348,48.272,159.745
C04989=1027.092,397.943,-147.556,173.358,48.274,159.747
C04990=1027.102,398.188,-147.600,173.369,48.277,159.749
C04991=1027.112,398.435,-147.644,173.379,48.279,159.751
C04992=1027.122,398.680,-147.689,173.389,48.281,159.753
C04993=1027.132,398.927,-147.733,173.400,48.283,159.755
C04994=1027.142,399.172,-147.778,173.410,48.287,159.758
C04995=1027.151,399.418,-147.822,173.421,48.289,159.760
C04996=1027.162,399.663,-147.866,173.431,48.291,159.762
C04997=1027.171,399.910,-147.910,173.441,48.294,159.764
C04998=1027.181,400.155,-147.955,173.452,48.296,159.766
C04999=1027.191,400.401,-148.000,173.463,48.299,159.769
C05000=1027.202,400.647,-148.045,173.474,48.301,159.771
C05001=1027.211,400.892,-148.089,173.484,48.304,159.773
C05002=1027.221,401.138,-148.134,173.495,48.307,159.775
C05003=1027.230,401.384,-148.178,173.506,48.309,159.777
C05004=1027.241,401.630,-148.224,173.517,48.312,159.780
C05005=1027.251,401.875,-148.268,173.527,48.315,159.782
C05006=1027.261,402.121,-148.313,173.538,48.317,159.784
C05007=1027.271,402.367,-148.358,173.549,48.320,159.787
C05008=1027.281,402.612,-148.403,173.560,48.322,159.789
C05009=1027.291,402.857,-148.448,173.571,48.325,159.791
C05010=1027.301,403.103,-148.493,173.582,48.328,159.793
C05011=1027.311,403.349,-148.538,173.592,48.331,159.796
C05012=1027.322,403.595,-148.584,173.603,48.334,159.798
C05013=1027.331,403.840,-148.629,173.614,48.336,159.800
C05014=1027.342,404.086,-148.674,173.625,48.339,159.803
C05015=1027.352,404.331,-148.720,173.636,48.342,159.805
C05016=1027.362,404.577,-148.765,173.647,48.345,159.807
C05017=1027.372,404.822,-148.810,173.659,48.348,159.810
C05018=1027.382,405.068,-148.856,173.670,48.351,159.812
C05019=1027.393,405.314,-148.902,173.681,48.353,159.815
C05020=1027.403,405.560,-148.946,173.692,48.356,159.817
C05021=1027.413,405.805,-148.992,173.704,48.360,159.820
C05022=1027.423,406.050,-149.038,173.715,48.362,159.822
C05023=1027.434,406.296,-149.083,173.726,48.365,159.824
C05024=1027.444,406.542,-149.129,173.737,48.368,159.827
C05025=1027.455,406.787,-149.175,173.748,48.371,159.829
C05026=1027.465,407.032,-149.220,173.761,48.374,159.832
C05027=1027.475,407.279,-149.266,173.772,48.377,159.834
C05028=1027.486,407.524,-149.311,173.783,48.380,159.837
C05029=1027.496,407.770,-149.357,173.795,48.383,159.839
C05030=1027.507,408.015,-149.403,173.806,48.386,159.842
C05031=1027.518,408.261,-149.449,173.818,48.389,159.844
C05032=1027.528,408.507,-149.495,173.830,48.392,159.847
C05033=1027.539,408.752,-149.541,173.841,48.395,159.849
C05034=1027.550,408.998,-149.587,173.853,48.398,159.852
C05035=1027.560,409.243,-149.633,173.865,48.401,159.854
C05036=1027.572,409.533,-149.687,173.878,48.405,159.857
C05037=1027.585,409.822,-149.741,173.892,48.409,159.860
C05038=1027.598,410.113,-149.796,173.906,48.412,159.863
C05039=1027.610,410.402,-149.852,173.920,48.416,159.866
C05040=1027.621,410.648,-149.898,173.932,48.419,159.869
C05041=1027.632,410.893,-149.944,173.944,48.422,159.872
C05042=1027.642,411.138,-149.991,173.956,48.426,159.874
C05043=1027.653,411.383,-150.037,173.968,48.429,159.877
C05044=1027.664,411.628,-150.084,173.980,48.432,159.879
C05045=1027.674,411.875,-150.131,173.992,48.436,159.882
C05046=1027.685,412.120,-150.177,174.004,48.439,159.885
C05047=1027.696,412.365,-150.224,174.016,48.443,159.888
C05048=1027.706,412.610,-150.271,174.028,48.446,159.890
C05049=1027.717,412.857,-150.318,174.040,48.450,159.893
C05050=1027.728,413.102,-150.364,174.053,48.452,159.896
C05051=1027.738,413.347,-150.411,174.066,48.456,159.898
C05052=1027.750,413.592,-150.458,174.077,48.459,159.901
C05053=1027.761,413.837,-150.505,174.090,48.463,159.904
C05054=1027.771,414.083,-150.552,174.102,48.466,159.907
C05055=1027.783,414.328,-150.599,174.114,48.470,159.910
C05056=1027.794,414.573,-150.647,174.127,48.473,159.912
C05057=1027.805,414.818,-150.694,174.139,48.477,159.915
C05058=1027.816,415.064,-150.741,174.152,48.480,159.918
C05059=1027.827,415.309,-150.788,174.164,48.483,159.921
C05060=1027.838,415.555,-150.836,174.177,48.487,159.923
C05061=1027.849,415.800,-150.883,174.189,48.491,159.926
C05062=1027.861,416.045,-150.930,174.202,48.494,159.929
C05063=1027.872,416.291,-150.978,174.215,48.498,159.932
C05064=1027.883,416.536,-151.025,174.228,48.502,159.935
C05065=1027.894,416.781,-151.073,174.241,48.505,159.938
C05066=1027.905,417.026,-151.121,174.254,48.509,159.941
C05067=1027.916,417.271,-151.168,174.266,48.513,159.944
C05068=1027.927,417.517,-151.216,174.279,48.516,159.946
C05069=1027.939,417.762,-151.264,174.292,48.520,159.949
C05070=1027.949,418.007,-151.312,174.305,48.524,159.952
C05071=1027.961,418.252,-151.359,174.318,48.528,159.955
C05072=1027.972,418.497,-151.408,174.331,48.532,159.958
C05073=1027.983,418.742,-151.456,174.344,48.535,159.961
C05074=1027.995,418.987,-151.504,174.357,48.539,159.964
C05075=1028.006,419.233,-151.552,174.370,48.543,159.967
C05076=1028.017,419.478,-151.600,174.383,48.547,159.970
C05077=1028.029,419.722,-151.648,174.396,48.550,159.973
C05078=1028.040,419.968,-151.696,174.410,48.554,159.976
C05079=1028.052,420.213,-151.744,174.424,48.558,159.979
C05080=1028.063,420.458,-151.793,174.437,48.562,159.983
C05081=1028.075,420.703,-151.841,174.450,48.566,159.986
C05082=1028.086,420.949,-151.889,174.463,48.570,159.989
C05083=1028.098,421.193,-151.938,174.478,48.574,159.992
C05084=1028.110,421.439,-151.986,174.491,48.578,159.995
C05085=1028.121,421.683,-152.035,174.504,48.582,159.998
C05086=1028.133,421.928,-152.082,174.517,48.586,160.001
C05087=1028.144,422.173,-152.131,174.532,48.590,160.005
C05088=1028.156,422.418,-152.181,174.545,48.594,160.008
C05089=1028.167,422.664,-152.229,174.560,48.598,160.011
C05090=1028.180,422.908,-152.278,174.573,48.602,160.014
C05091=1028.191,423.153,-152.327,174.586,48.606,160.017
C05092=1028.203,423.398,-152.376,174.601,48.610,160.020
C05093=1028.214,423.643,-152.425,174.614,48.614,160.024
C05094=1028.226,423.888,-152.474,174.629,48.618,160.027
C05095=1028.239,424.133,-152.523,174.642,48.623,160.030
C05096=1028.250,424.360,-152.569,174.655,48.626,160.033
C05097=1028.260,424.588,-152.614,174.668,48.630,160.036
C05098=1028.271,424.814,-152.661,174.682,48.634,160.039
C05099=1028.283,425.042,-152.705,174.695,48.638,160.043
C05100=1028.293,425.269,-152.752,174.708,48.642,160.046
C05101=1028.304,425.496,-152.798,174.722,48.646,160.049
C05102=1028.315,425.723,-152.843,174.735,48.650,160.052
C05103=1028.327,425.950,-152.889,174.748,48.654,160.055
C05104=1028.339,426.194,-152.938,174.762,48.658,160.058
C05105=1028.351,426.439,-152.988,174.777,48.663,160.062
C05106=1028.363,426.684,-153.038,174.791,48.667,160.065
C05107=1028.375,426.928,-153.088,174.806,48.672,160.069
C05108=1028.387,427.174,-153.137,174.820,48.676,160.072
C05109=1028.399,427.418,-153.187,174.835,48.681,160.075
C05110=1028.411,427.663,-153.237,174.849,48.685,160.079
C05111=1028.423,427.907,-153.287,174.864,48.689,160.082
C05112=1028.435,428.152,-153.337,174.879,48.694,160.086
C05113=1028.448,428.397,-153.387,174.894,48.698,160.089
C05114=1028.459,428.642,-153.438,174.908,48.702,160.093
C05115=1028.471,428.886,-153.488,174.923,48.707,160.096
C05116=1028.483,429.131,-153.538,174.938,48.712,160.100
C05117=1028.496,429.375,-153.588,174.953,48.716,160.103
C05118=1028.508,429.620,-153.639,174.968,48.721,160.107
C05119=1028.520,429.865,-153.689,174.983,48.725,160.111
C05120=1028.533,430.109,-153.739,174.999,48.730,160.114
C05121=1028.545,430.354,-153.790,175.014,48.735,160.118
C05122=1028.558,430.599,-153.840,175.029,48.739,160.122
C05123=1028.570,430.843,-153.890,175.044,48.744,160.125
C05124=1028.583,431.088,-153.942,175.060,48.749,160.129
C05125=1028.596,431.333,-153.992,175.076,48.753,160.133
C05126=1028.608,431.577,-154.043,175.091,48.758,160.136
C05127=1028.621,431.821,-154.093,175.106,48.763,160.140
C05128=1028.633,432.066,-154.143,175.122,48.768,160.144
C05129=1028.647,432.311,-154.195,175.137,48.773,160.148
C05130=1028.659,432.555,-154.245,175.153,48.778,160.151
C05131=1028.672,432.799,-154.296,175.169,48.782,160.155
C05132=1028.685,433.044,-154.347,175.184,48.787,160.159
C05133=1028.697,433.289,-154.399,175.200,48.792,160.163
C05134=1028.710,433.534,-154.450,175.216,48.797,160.166
C05135=1028.723,433.778,-154.501,175.232,48.801,160.170
C05136=1028.740,434.113,-154.572,175.254,48.808,160.176
C05137=1028.759,434.447,-154.642,175.276,48.815,160.181
C05138=1028.776,434.783,-154.712,175.298,48.822,160.186
C05139=1028.794,435.118,-154.783,175.321,48.828,160.192
C05140=1028.807,435.362,-154.835,175.337,48.834,160.196
C05141=1028.820,435.607,-154.886,175.353,48.839,160.200
C05142=1028.832,435.851,-154.939,175.370,48.844,160.204
C05143=1028.846,436.095,-154.991,175.386,48.849,160.208
C05144=1028.859,436.339,-155.042,175.403,48.854,160.212
C05145=1028.872,436.584,-155.095,175.420,48.860,160.216
C05146=1028.885,436.828,-155.146,175.436,48.865,160.220
C05147=1028.899,437.072,-155.198,175.453,48.870,160.224
C05148=1028.912,437.317,-155.251,175.470,48.875,160.228
C05149=1028.924,437.560,-155.302,175.486,48.880,160.232
C05150=1028.938,437.805,-155.354,175.503,48.885,160.236
C05151=1028.951,438.049,-155.407,175.520,48.891,160.240
C05152=1028.965,438.293,-155.459,175.537,48.896,160.245
C05153=1028.978,438.537,-155.511,175.554,48.901,160.249
C05154=1028.991,438.782,-155.564,175.571,48.906,160.253
C05155=1029.005,439.025,-155.616,175.588,48.912,160.257
C05156=1029.020,439.296,-155.675,175.607,48.918,160.262
C05157=1029.035,439.567,-155.733,175.627,48.924,160.267
C05158=1029.049,439.836,-155.791,175.646,48.930,160.271
C05159=1029.065,440.107,-155.850,175.665,48.936,160.276
C05160=1029.078,440.351,-155.903,175.683,48.941,160.280
C05161=1029.092,440.594,-155.956,175.700,48.947,160.285
C05162=1029.105,440.839,-156.009,175.718,48.952,160.289
C05163=1029.119,441.082,-156.062,175.735,48.958,160.293
C05164=1029.132,441.326,-156.115,175.754,48.963,160.298
C05165=1029.147,441.571,-156.168,175.771,48.969,160.302
C05166=1029.161,441.814,-156.221,175.789,48.974,160.307
C05167=1029.174,442.058,-156.274,175.807,48.980,160.311
C05168=1029.188,442.302,-156.327,175.825,48.985,160.316
C05169=1029.202,442.546,-156.381,175.843,48.991,160.320
C05170=1029.216,442.789,-156.434,175.861,48.997,160.325
C05171=1029.230,443.033,-156.488,175.879,49.002,160.329
C05172=1029.244,443.276,-156.541,175.898,49.008,160.334
C05173=1029.259,443.519,-156.593,175.916,49.013,160.338
C05174=1029.275,443.762,-156.646,175.934,49.019,160.343
C05175=1029.291,444.006,-156.697,175.952,49.024,160.347
C05176=1029.307,444.249,-156.748,175.972,49.029,160.352
C05177=1029.323,444.493,-156.799,175.990,49.035,160.356
C05178=1029.341,444.737,-156.850,176.009,49.039,160.360
C05179=1029.359,444.981,-156.900,176.028,49.045,160.365
C05180=1029.377,445.225,-156.949,176.047,49.050,160.369
C05181=1029.395,445.469,-156.999,176.066,49.055,160.374
C05182=1029.415,445.712,-157.048,176.085,49.059,160.378
C05183=1029.435,445.957,-157.096,176.104,49.064,160.383
C05184=1029.455,446.201,-157.144,176.124,49.068,160.387
C05185=1029.476,446.445,-157.192,176.143,49.073,160.392
C05186=1029.497,446.690,-157.239,176.162,49.078,160.396
C05187=1029.518,446.934,-157.286,176.182,49.082,160.400
C05188=1029.541,447.179,-157.332,176.201,49.087,160.405
C05189=1029.563,447.423,-157.379,176.221,49.091,160.409
C05190=1029.586,447.668,-157.425,176.241,49.095,160.414
C05191=1029.609,447.913,-157.470,176.261,49.099,160.418
C05192=1029.634,448.158,-157.515,176.281,49.104,160.422
C05193=1029.658,448.403,-157.558,176.301,49.108,160.427
C05194=1029.682,448.647,-157.603,176.321,49.112,160.431
C05195=1029.708,448.893,-157.646,176.341,49.115,160.435
C05196=1029.734,449.138,-157.690,176.361,49.120,160.440
C05197=1029.761,449.383,-157.732,176.382,49.123,160.444
C05198=1029.788,449.628,-157.775,176.402,49.127,160.449
C05199=1029.815,449.873,-157.817,176.422,49.131,160.453
C05200=1029.843,450.119,-157.859,176.443,49.134,160.457
C05201=1029.871,450.364,-157.899,176.464,49.138,160.462
C05202=1029.900,450.609,-157.940,176.485,49.142,160.466
C05203=1029.929,450.854,-157.980,176.505,49.145,160.470
C05204=1029.958,451.100,-158.021,176.527,49.148,160.475
C05205=1029.990,451.345,-158.061,176.548,49.151,160.479
C05206=1030.020,451.591,-158.099,176.569,49.154,160.483
C05207=1030.051,451.837,-158.138,176.590,49.158,160.488
C05208=1030.083,452.082,-158.177,176.612,49.161,160.492
C05209=1030.115,452.328,-158.214,176.633,49.164,160.496
C05210=1030.147,452.573,-158.252,176.655,49.167,160.501
C05211=1030.181,452.818,-158.289,176.677,49.169,160.505
C05212=1030.215,453.065,-158.326,176.698,49.173,160.509
C05213=1030.248,453.311,-158.363,176.720,49.176,160.514
C05214=1030.283,453.556,-158.398,176.742,49.178,160.518
C05215=1030.327,453.861,-158.442,176.769,49.182,160.523
C05216=1030.048,453.933,-158.776,176.773,49.244,160.543
C05217=1030.010,453.669,-158.739,176.749,49.241,160.539
C05218=1029.976,453.424,-158.703,176.726,49.239,160.535
C05219=1029.941,453.178,-158.667,176.705,49.236,160.530
C05220=1029.908,452.931,-158.630,176.683,49.233,160.526
C05221=1029.874,452.687,-158.594,176.662,49.231,160.522
C05222=1029.841,452.440,-158.556,176.640,49.227,160.517
C05223=1029.809,452.195,-158.518,176.618,49.224,160.513
C05224=1029.777,451.949,-158.480,176.597,49.222,160.509
C05225=1029.746,451.704,-158.441,176.575,49.219,160.504
C05226=1029.714,451.458,-158.403,176.554,49.216,160.500
C05227=1029.684,451.212,-158.363,176.533,49.213,160.496
C05228=1029.654,450.967,-158.323,176.511,49.209,160.491
C05229=1029.624,450.722,-158.283,176.490,49.206,160.487
C05230=1029.595,450.477,-158.243,176.470,49.203,160.483
C05231=1029.566,450.231,-158.202,176.449,49.199,160.478
C05232=1029.538,449.986,-158.161,176.428,49.196,160.474
C05233=1029.510,449.740,-158.119,176.408,49.192,160.470
C05234=1029.484,449.495,-158.077,176.387,49.188,160.465
C05235=1029.457,449.250,-158.034,176.366,49.185,160.461
C05236=1029.431,449.005,-157.991,176.346,49.181,160.457
C05237=1029.405,448.759,-157.948,176.325,49.178,160.452
C05238=1029.380,448.515,-157.904,176.305,49.173,160.448
C05239=1029.356,448.270,-157.860,176.286,49.170,160.444
C05240=1029.331,448.025,-157.815,176.265,49.166,160.439
C05241=1029.307,447.780,-157.770,176.245,49.161,160.435
C05242=1029.284,447.536,-157.725,176.225,49.158,160.430
C05243=1029.261,447.291,-157.679,176.205,49.153,160.426
C05244=1029.239,447.047,-157.633,176.186,49.149,160.422
C05245=1029.217,446.802,-157.585,176.166,49.145,160.417
C05246=1029.195,446.557,-157.539,176.147,49.140,160.413
C05247=1029.175,446.314,-157.491,176.127,49.136,160.408
C05248=1029.154,446.069,-157.444,176.108,49.131,160.404
C05249=1029.134,445.825,-157.396,176.089,49.127,160.400
C05250=1029.114,445.581,-157.347,176.069,49.122,160.395
C05251=1029.095,445.337,-157.297,176.050,49.117,160.391
C05252=1029.077,445.093,-157.248,176.032,49.112,160.386
C05253=1029.058,444.849,-157.198,176.013,49.108,160.382
C05254=1029.041,444.605,-157.148,175.994,49.103,160.377
C05255=1029.024,444.362,-157.098,175.974,49.097,160.373
C05256=1029.007,444.118,-157.047,175.956,49.092,160.368
C05257=1028.991,443.873,-156.995,175.938,49.087,160.364
C05258=1028.976,443.630,-156.944,175.919,49.082,160.359
C05259=1028.960,443.387,-156.891,175.900,49.077,160.355
C05260=1028.945,443.144,-156.838,175.882,49.072,160.351
C05261=1028.932,442.901,-156.785,175.864,49.066,160.346
C05262=1028.917,442.658,-156.732,175.845,49.060,160.341
C05263=1028.903,442.413,-156.679,175.827,49.055,160.337
C05264=1028.890,442.170,-156.625,175.810,49.049,160.333
C05265=1028.876,441.926,-156.572,175.792,49.043,160.328
C05266=1028.861,441.682,-156.519,175.773,49.038,160.324
C05267=1028.848,441.438,-156.466,175.755,49.033,160.319
C05268=1028.834,441.195,-156.413,175.738,49.027,160.315
C05269=1028.820,440.950,-156.359,175.720,49.022,160.311
C05270=1028.807,440.707,-156.307,175.702,49.017,160.306
C05271=1028.793,440.463,-156.254,175.685,49.011,160.302
C05272=1028.780,440.219,-156.201,175.667,49.006,160.297
C05273=1028.764,439.947,-156.143,175.648,49.000,160.293
C05274=1028.750,439.677,-156.083,175.629,48.994,160.288
C05275=1028.734,439.405,-156.025,175.609,48.988,160.283
C05276=1028.719,439.135,-155.966,175.590,48.982,160.279
C05277=1028.706,438.890,-155.914,175.572,48.977,160.274
C05278=1028.692,438.646,-155.861,175.555,48.972,160.270
C05279=1028.680,438.402,-155.809,175.538,48.966,160.266
C05280=1028.666,438.158,-155.757,175.521,48.961,160.262
C05281=1028.652,437.914,-155.704,175.504,48.956,160.257
C05282=1028.639,437.669,-155.652,175.487,48.951,160.253
C05283=1028.626,437.425,-155.600,175.470,48.946,160.249
C05284=1028.612,437.181,-155.548,175.454,48.941,160.245
C05285=1028.600,436.936,-155.496,175.437,48.936,160.241
C05286=1028.587,436.693,-155.444,175.420,48.930,160.237
C05287=1028.573,436.448,-155.392,175.403,48.925,160.233
C05288=1028.560,436.204,-155.340,175.387,48.921,160.229
C05289=1028.547,435.959,-155.288,175.370,48.915,160.225
C05290=1028.534,435.716,-155.236,175.354,48.910,160.221
C05291=1028.520,435.472,-155.184,175.337,48.906,160.217
C05292=1028.508,435.226,-155.133,175.321,48.900,160.213
C05293=1028.495,434.983,-155.081,175.304,48.896,160.209
C05294=1028.482,434.738,-155.030,175.288,48.891,160.205
C05295=1028.469,434.494,-154.978,175.272,48.886,160.201
C05296=1028.456,434.249,-154.927,175.256,48.881,160.197
C05297=1028.443,434.005,-154.875,175.240,48.876,160.193
C05298=1028.430,433.761,-154.824,175.224,48.871,160.190
C05299=1028.418,433.516,-154.773,175.208,48.866,160.186
C05300=1028.405,433.271,-154.721,175.192,48.862,160.182
C05301=1028.393,433.027,-154.671,175.176,48.857,160.178
C05302=1028.380,432.783,-154.620,175.160,48.852,160.174
C05303=1028.367,432.538,-154.569,175.145,48.848,160.171
C05304=1028.354,432.294,-154.518,175.129,48.843,160.167
C05305=1028.341,432.049,-154.467,175.113,48.838,160.163
C05306=1028.328,431.805,-154.416,175.097,48.834,160.159
C05307=1028.316,431.560,-154.365,175.082,48.828,160.155
C05308=1028.303,431.316,-154.315,175.066,48.824,160.152
C05309=1028.291,431.071,-154.264,175.051,48.820,160.148
C05310=1028.278,430.827,-154.213,175.036,48.815,160.144
C05311=1028.266,430.582,-154.163,175.021,48.810,160.141
C05312=1028.253,430.337,-154.112,175.005,48.806,160.137
C05313=1028.240,430.093,-154.062,174.990,48.801,160.134
C05314=1028.228,429.848,-154.012,174.975,48.797,160.130
C05315=1028.215,429.604,-153.961,174.960,48.792,160.126
C05316=1028.203,429.359,-153.911,174.945,48.788,160.123
C05317=1028.191,429.115,-153.861,174.929,48.783,160.119
C05318=1028.179,428.870,-153.810,174.914,48.779,160.116
C05319=1028.166,428.626,-153.760,174.899,48.774,160.112
C05320=1028.154,428.381,-153.710,174.884,48.770,160.109
C05321=1028.137,428.027,-153.638,174.863,48.764,160.104
C05322=1028.120,427.673,-153.566,174.841,48.757,160.099
C05323=1028.102,427.320,-153.494,174.820,48.751,160.093
C05324=1028.085,426.966,-153.422,174.799,48.745,160.089
C05325=1028.072,426.721,-153.372,174.785,48.740,160.085
C05326=1028.061,426.477,-153.322,174.770,48.736,160.082
C05327=1028.049,426.232,-153.273,174.755,48.732,160.078
C05328=1028.036,425.987,-153.222,174.742,48.727,160.075
C05329=1028.025,425.768,-153.179,174.728,48.724,160.072
C05330=1028.015,425.549,-153.134,174.715,48.720,160.069
C05331=1028.004,425.330,-153.090,174.702,48.716,160.066
C05332=1027.993,425.110,-153.046,174.690,48.712,160.063
C05333=1027.983,424.891,-153.001,174.677,48.709,160.060
C05334=1027.972,424.672,-152.958,174.664,48.705,160.057
C05335=1027.961,424.452,-152.913,174.652,48.701,160.054
C05336=1027.951,424.232,-152.869,174.639,48.698,160.051
C05337=1027.939,423.988,-152.821,174.626,48.694,160.048
C05338=1027.927,423.743,-152.772,174.611,48.690,160.045
C05339=1027.915,423.497,-152.722,174.596,48.686,160.041
C05340=1027.904,423.253,-152.673,174.583,48.682,160.038
C05341=1027.892,423.008,-152.624,174.570,48.677,160.035
C05342=1027.880,422.764,-152.576,174.555,48.674,160.032
C05343=1027.868,422.518,-152.526,174.542,48.669,160.028
C05344=1027.857,422.273,-152.478,174.528,48.666,160.025
C05345=1027.846,422.028,-152.429,174.514,48.662,160.022
C05346=1027.834,421.784,-152.381,174.500,48.658,160.019
C05347=1027.822,421.538,-152.332,174.487,48.654,160.016
C05348=1027.810,421.293,-152.284,174.473,48.650,160.013
C05349=1027.799,421.048,-152.235,174.459,48.646,160.010
C05350=1027.787,420.803,-152.186,174.446,48.642,160.007
C05351=1027.775,420.558,-152.139,174.433,48.638,160.003
C05352=1027.764,420.313,-152.090,174.419,48.634,160.000
C05353=1027.752,420.068,-152.042,174.405,48.631,159.997
C05354=1027.741,419.823,-151.994,174.392,48.627,159.994
C05355=1027.730,419.577,-151.945,174.379,48.623,159.991
C05356=1027.718,419.332,-151.898,174.366,48.619,159.988
C05357=1027.707,419.087,-151.849,174.353,48.615,159.985
